		MesCP_Read					: BOOL := TRUE;	(* Read function enable *)
		MesCP_Write					: BOOL := TRUE;	(* Write function enable *)
                 
END_VAR

METHOD M_AlarmManagement
//////////////////
// Digiware measurement tool alarm and warning management
/////////////////

VAR 
	
END_VAR
END_METHOD

METHOD M_CP
//////////////////
//  Emulator
/////////////////

VAR 
	// Method local variables (reinitialized at each cycle) 
	
END_VAR
Trig_Cmd_Read(CLK:=IN_CmdToggleRead);

IF Trig_Cmd_Read.Q THEN
	IN_CmdToggleRead := FALSE;
	MesCP_Read := NOT MesCP_Read;
END_IF
END_METHOD

METHOD M_Execute
//////////////////
//  Method Calls 
/////////////////
VAR 
	// Method local variables (reinitialized at each cycle) 
	// EMULATOR

	
END_VAR
// READING AND WRITING CLOCK //
	TP1(IN:=NOT TP1.Q , PT:= ParamClockReadTime);
	ClockRead 		:= TP1.Q;

// PERMANENT CONDITIONS //
	M_CP() ; 
	
// METHODS CALLS //
	IF bInit THEN
		M_Init() ; 
		bInit					:= FALSE ; 
	ELSIF CmdInit_G OR IN_CmdReset_L THEN 
		bInit:= TRUE ;		
	END_IF

	M_Read() ; 
	M_AlarmManagement();
END_METHOD

METHOD M_Init
VAR 

END_VAR
END_METHOD

METHOD M_Read
//////////////////
//  Read Modbus Variable for PCS . 
/////////////////
VAR 
	// Method local variables (reinitialized at each cycle) 
	
END_VAR
END_METHOD

END_FUNCTION_BLOCK

// ---- 01_Equipement_Library/Operation Meter/FB_PM_A40.TcPOU
FUNCTION_BLOCK FB_PM_A40 EXTENDS FB_PM_Base
//////////////////
// Measurement Solution based on Digiware, but access through PMS Socomec
//////////////////

VAR_INPUT PERSISTENT
	// Parameters of the Object (instance specific)
	{attribute 'OPC.UA.DA' := '1'}  
	ParamUnitID					: BYTE := 22; 										// (NA) All unit ID For the Device (I35 + 1 U20)                                                                    			
	{attribute 'OPC.UA.DA' := '1'}                                                                             			
	ParamIPAddress			   	: STRING := '192.168.20.15'; 						// (NA) IP Adress of D50 .
	{attribute 'OPC.UA.DA' := '1'} 
	ParamTCPPort				: UINT := 502;										// Modbus TCP Port


END_VAR

VAR_OUTPUT
	//Child objects
	
END_VAR
VAR
	//M_ALARMMANAGEMENT VARIABLES//
		
	//M_READ VARIABLES//
		FB_ModbusRead_I1			: ARRAY[1..2] OF  FB_ModbusRead ; 				// (NA) FB for Modbus Reading
	                                                                                    	
		MesBlock1_Temp 				: ARRAY[1..2] 	OF ARRAY[0..124] OF WORD;		//(NA) Temporary Block with multiple modbus reading (U30 + I35)
		MesModbusReadAlarm 		  	: ARRAY[1..2] OF BOOL ; 						// (NA) Modbus Read Alarm for communication 
		
		
		MesModbusAlarmCode			: ARRAY[1..2] OF UDINT;							// (NA) Modbus Read Alarm Code	
		
	//M_INIT VARIABLES //
		
	// M_EXECUTE VARIABLES //
		   	MesDataExd AT %Q*			: PM_Standard ;               


 
END_VAR

METHOD M_AlarmManagement
//////////////////
// Digiware measurement tool alarm and warning management
/////////////////

VAR 
	// Method local variables (reinitialized at each cycle) 
	FB_AlarmCodeManager			: FB_AlarmCodeManager ; 
	
	KK							: BYTE ;		// For loop
	
	CMWarning					: BOOL;			// At least one Digiware device in Alarm
	CMAlarm						: BOOL;			// At least one Digiware device in Alarm
	
END_VAR
// COMMUNICATION // 

		CMWarning 		:= MesModbusReadAlarm[1] ;
		CMAlarm			:= MesModbusReadAlarm[1];
		
	// Warning
	MesWarningCom 		:= CMWarning ; 											// LOC with at least one Digiware module
	//Alarm
	TON_ComAlarm(IN:= CMAlarm, PT:= ParamTempoComAlarm, Q=>MesDataExd.MesData.MesAlarmCom) ;	 	// D50 LOC

// ALARM CODE //
	FB_AlarmCodeManager(
		bAlarm1			:=MesDataExd.MesData.MesAlarmCom , 					// Communication Alarm  #COM
		bAlarm2			:=FALSE, 									// 
		bAlarm3			:=FALSE, 									// 
		bAlarm4			:=FALSE, 									// 
		bAlarm5			:=FALSE, 									//
		bAlarm6			:=FALSE,                                    //
		bAlarm7			:=FALSE,                                    //
		bAlarm8			:=FALSE, 									//
		bAlarm9			:=FALSE,                                    //
		bAlarm10		:=FALSE,                                    //
		bAlarm11		:=FALSE, 									//
		bAlarm12		:=FALSE,                                    //
		bAlarm13		:=FALSE,                                    //
		bAlarm14		:=FALSE, 									//
		bAlarm15		:= FALSE , 									// 						 
		wAlarmCode		=>MesDataExd.MesData.MesAlarmCode);

// WARNING CODE //
	FB_AlarmCodeManager(		
		bAlarm1			:= MesWarningCom,				// Communication warning  #COM
		bAlarm2			:=FALSE, 						// 
		bAlarm3			:=FALSE, 						// 
		bAlarm4			:=FALSE, 						// 
		bAlarm5			:=FALSE, 						//
		bAlarm6			:=FALSE,                        //
		bAlarm7			:=FALSE,                        //
		bAlarm8			:=FALSE,                        //
		bAlarm9			:=FALSE,                        //
		bAlarm10		:=FALSE,                        //
		bAlarm11		:=FALSE,                        //
		bAlarm12		:=FALSE,                        //
		bAlarm13		:=FALSE,                        //
		bAlarm14		:=FALSE,                        //
		bAlarm15		:=FALSE,                        //
		wAlarmCode		=>MesDataExd.MesData.MesWarningCode);
END_METHOD

METHOD M_Read
//////////////////
//  Read Modbus Variable for PCS . 
/////////////////
VAR 
	// Method local variables (reinitialized at each cycle) 
	MW 					: FB_MergeWordsToDint; 
	KK					: BYTE;  						// FOR Loop 

	Pinterm				: REAL;
	Pinterm1			: REAL;
	Pinterm2			: REAL;
	Pinterm3			: REAL;
	Iinterm1			: REAL;
	Iinterm2			: REAL;
	Iinterm3			: REAL;
	IInterm				: REAL;
	QInterm1			: REAL;
	QInterm2			: REAL;
	QInterm3			: REAL;
	QInterm				: REAL;
	SInterm				: REAL;
END_VAR
//INITIALIZING MODBUS REQUESTS //
	FOR KK:=1 TO 2 DO
		FB_ModbusRead_I1[KK](Reset:= CmdClearFault_G ,sIPAddr:=ParamIPAddress, tTimeout:= ParamTimeout, 	nTCPport := ParamTCPPort	);
	
	END_FOR 

// CP-Read / Write 

MesDataExd.MesData.MesCP_Read := MesCP_Read ; 

IF MesCP_Read  THEN		
// MODBUS REQUEST//
	FB_ModbusRead_I1[1](
		nQuantity		:= 89, 
		nMBAddr			:= 16#4800, 
		nUnitID			:= ParamUnitID,
		cbLength		:= SIZEOF(MesBlock1_Temp[1]) , 
		pDestAddr		:= ADR(MesBlock1_Temp[1]) ,
		ClockRead		:=  MesCP_Read AND ClockRead ,
		ModbusReadAlarm	=>	MesModbusReadAlarm[1]);
		
		
		
	FB_ModbusRead_I1[2](
		nQuantity		:= 54, 
		nMBAddr			:= 16#4D80, 
		nUnitID			:= ParamUnitID,
		cbLength		:= SIZEOF(MesBlock1_Temp[2]) , 
		pDestAddr		:= ADR(MesBlock1_Temp[2]) ,
		ClockRead		:=  MesCP_Read AND ClockRead ,
		ModbusReadAlarm	=>	MesModbusReadAlarm[2]);		
		
		
// PROPERTIES UPDATE // 
	
	// Block2
	MW(WORD_STRONG:= MesBlock1_Temp[1][4], WORD_WEAK := MesBlock1_Temp[1][5],SIGNED:=FALSE, FIX:=2 , SIZE:=2, VAR_OUT := MesDataExd.MesData.MesV);	
	MW(WORD_STRONG:= MesBlock1_Temp[1][6], WORD_WEAK := MesBlock1_Temp[1][7],SIGNED:=FALSE, FIX:=2 , SIZE:=2, VAR_OUT := MesDataExd.MesData.MesU);	
	MW(WORD_STRONG:= MesBlock1_Temp[1][8], WORD_WEAK := MesBlock1_Temp[1][9],SIGNED:=FALSE, FIX:=3 , SIZE:=2, VAR_OUT := MesDataExd.MesData.MesI);	
	MW(WORD_STRONG:= MesBlock1_Temp[1][10], WORD_WEAK := MesBlock1_Temp[1][11],SIGNED:=FALSE, FIX:=3 , SIZE:=2, VAR_OUT := MesDataExd.MesData.MesFreq);	
	MW(WORD_STRONG:= MesBlock1_Temp[1][12], WORD_WEAK := MesBlock1_Temp[1][13],SIGNED:=FALSE, FIX:=2 , SIZE:=2, VAR_OUT := MesDataExd.MesData.MesV1);	
	MW(WORD_STRONG:= MesBlock1_Temp[1][14], WORD_WEAK := MesBlock1_Temp[1][15],SIGNED:=FALSE, FIX:=2 , SIZE:=2, VAR_OUT := MesDataExd.MesData.MesV2);	
	MW(WORD_STRONG:= MesBlock1_Temp[1][16], WORD_WEAK := MesBlock1_Temp[1][17],SIGNED:=FALSE, FIX:=2 , SIZE:=2, VAR_OUT := MesDataExd.MesData.MesV3);	
	MW(WORD_STRONG:= MesBlock1_Temp[1][20], WORD_WEAK := MesBlock1_Temp[1][21],SIGNED:=FALSE, FIX:=2 , SIZE:=2, VAR_OUT := MesDataExd.MesData.MesU12);	
	MW(WORD_STRONG:= MesBlock1_Temp[1][22], WORD_WEAK := MesBlock1_Temp[1][23],SIGNED:=FALSE, FIX:=2 , SIZE:=2, VAR_OUT := MesDataExd.MesData.MesU23);	
	MW(WORD_STRONG:= MesBlock1_Temp[1][24], WORD_WEAK := MesBlock1_Temp[1][25],SIGNED:=FALSE, FIX:=2 , SIZE:=2, VAR_OUT := MesDataExd.MesData.MesU31);	
	MW(WORD_STRONG:= MesBlock1_Temp[1][26], WORD_WEAK := MesBlock1_Temp[1][27],SIGNED:=FALSE, FIX:=3 , SIZE:=2, VAR_OUT := MesDataExd.MesData.MesI1);	
	MW(WORD_STRONG:= MesBlock1_Temp[1][28], WORD_WEAK := MesBlock1_Temp[1][29],SIGNED:=FALSE, FIX:=3 , SIZE:=2, VAR_OUT := MesDataExd.MesData.MesI2);	
	MW(WORD_STRONG:= MesBlock1_Temp[1][30], WORD_WEAK := MesBlock1_Temp[1][31],SIGNED:=FALSE, FIX:=3 , SIZE:=2, VAR_OUT := MesDataExd.MesData.MesI3);
	MW(WORD_STRONG:= MesBlock1_Temp[1][44], WORD_WEAK := MesBlock1_Temp[1][45],SIGNED:=TRUE, FIX:=3 , SIZE:=2, VAR_OUT := MesDataExd.MesData.MesP);	
	MW(WORD_STRONG:= MesBlock1_Temp[1][46], WORD_WEAK := MesBlock1_Temp[1][47],SIGNED:=TRUE, FIX:=3 , SIZE:=2, VAR_OUT := MesDataExd.MesData.MesQ);	
	MW(WORD_STRONG:= MesBlock1_Temp[1][52], WORD_WEAK := MesBlock1_Temp[1][53],SIGNED:=FALSE, FIX:=3 , SIZE:=2, VAR_OUT := MesDataExd.MesData.MesS);	
	MW(WORD_STRONG:= MesBlock1_Temp[1][54],SIGNED:=TRUE, FIX:=3 , SIZE:=1, VAR_OUT := MesDataExd.MesData.MesCosPhi);		
	MW(WORD_STRONG:= MesBlock1_Temp[1][56], WORD_WEAK := MesBlock1_Temp[1][57],SIGNED:=TRUE, FIX:=3 , SIZE:=2, VAR_OUT := MesDataExd.MesData.MesP1);	
	MW(WORD_STRONG:= MesBlock1_Temp[1][58], WORD_WEAK := MesBlock1_Temp[1][59],SIGNED:=TRUE, FIX:=3 , SIZE:=2, VAR_OUT := MesDataExd.MesData.MesP2);	
	MW(WORD_STRONG:= MesBlock1_Temp[1][60], WORD_WEAK := MesBlock1_Temp[1][61],SIGNED:=TRUE, FIX:=3 , SIZE:=2, VAR_OUT := MesDataExd.MesData.MesP3);	
	MW(WORD_STRONG:= MesBlock1_Temp[1][62], WORD_WEAK := MesBlock1_Temp[1][63],SIGNED:=TRUE, FIX:=3 , SIZE:=2, VAR_OUT := MesDataExd.MesData.MesQ1);	
	MW(WORD_STRONG:= MesBlock1_Temp[1][64], WORD_WEAK := MesBlock1_Temp[1][65],SIGNED:=TRUE, FIX:=3 , SIZE:=2, VAR_OUT := MesDataExd.MesData.MesQ2);	
	MW(WORD_STRONG:= MesBlock1_Temp[1][66], WORD_WEAK := MesBlock1_Temp[1][67],SIGNED:=TRUE, FIX:=3 , SIZE:=2, VAR_OUT := MesDataExd.MesData.MesQ3);		
	MW(WORD_STRONG:= MesBlock1_Temp[1][80], WORD_WEAK := MesBlock1_Temp[1][81],SIGNED:=FALSE, FIX:=3 , SIZE:=2, VAR_OUT := MesDataExd.MesData.MesS1);	
	MW(WORD_STRONG:= MesBlock1_Temp[1][82], WORD_WEAK := MesBlock1_Temp[1][83],SIGNED:=FALSE, FIX:=3 , SIZE:=2, VAR_OUT := MesDataExd.MesData.MesS2);	
	MW(WORD_STRONG:= MesBlock1_Temp[1][84], WORD_WEAK := MesBlock1_Temp[1][85],SIGNED:=FALSE, FIX:=3 , SIZE:=2, VAR_OUT := MesDataExd.MesData.MesS3);	
	MW(WORD_STRONG:= MesBlock1_Temp[1][86],SIGNED:=TRUE, FIX:=3 , SIZE:=1, VAR_OUT := MesDataExd.MesData.MesCosPhi1);	
	MW(WORD_STRONG:= MesBlock1_Temp[1][87],SIGNED:=TRUE, FIX:=3 , SIZE:=1, VAR_OUT := MesDataExd.MesData.MesCosPhi2);
	MW(WORD_STRONG:= MesBlock1_Temp[1][88],SIGNED:=TRUE, FIX:=3 , SIZE:=1, VAR_OUT := MesDataExd.MesData.MesCosPhi3);
	

	// energies 
	MW(WORD_STRONG:= MesBlock1_Temp[2][4], WORD_WEAK := MesBlock1_Temp[2][5],SIGNED:=FALSE, FIX:=4 , SIZE:=2, VAR_OUT := MesDataExd.MesData.MesEActCons);
	MW(WORD_STRONG:= MesBlock1_Temp[2][7], WORD_WEAK := MesBlock1_Temp[2][8],SIGNED:=FALSE, FIX:=4 , SIZE:=2, VAR_OUT := MesDataExd.MesData.MesEActProd);	
	MW(WORD_STRONG:= MesBlock1_Temp[2][10], WORD_WEAK := MesBlock1_Temp[2][11],SIGNED:=FALSE, FIX:=4 , SIZE:=2, VAR_OUT := MesDataExd.MesData.MesEReactCons);
	MW(WORD_STRONG:= MesBlock1_Temp[2][13], WORD_WEAK := MesBlock1_Temp[2][14],SIGNED:=FALSE, FIX:=4 , SIZE:=2, VAR_OUT := MesDataExd.MesData.MesEReactProd);
	

END_IF

// Evaluate 
	IF MesDataExd.MesData.MesP > 0.01 OR MesDataExd.MesData.MesP < -0.01 THEN
	MesDataExd.MesData.MesTanPhi := MesDataExd.MesData.MesQ /MesDataExd.MesData.MesP;
	ELSE
	MesDataExd.MesData.MesTanPhi := 0;
	END_IF
END_METHOD

END_FUNCTION_BLOCK

// ---- 01_Equipement_Library/Operation Meter/FB_PM_Digiware.TcPOU
FUNCTION_BLOCK FB_PM_Digiware EXTENDS FB_PM_Base
//////////////////
// Measurement Solution based on Digiware, but access through PMS Socomec
//////////////////

VAR_INPUT PERSISTENT
	// Parameters of the Object (instance specific) 
	ParamUnitID					: BYTE	 	;						// (NA) U30 unit ID
	ParamIPAddress			   	: STRING 	;							// (NA) IP Adress of D50 .
	ParamTCPPort				: UINT 		;
	ParamInvertPower			: BOOL		;
END_VAR

VAR_OUTPUT
	//Child objects
	
END_VAR
VAR
	//M_ALARMMANAGEMENT VARIABLES//
		
	//M_READ VARIABLES//
		MesDataExd					: PM_DirisA40;
		
		ModbusRead					: ARRAY[1..5] OF FB_ModbusRead ; 			// (NA) FB for Modbus Reading
		MesBlock1_Temp 				: ARRAY[1..5] OF ARRAY[1..120] OF WORD;		//(NA) Temporary Block with multiple modbus reading (U30 + I35)
		
		
	//M_CP VARIABLES //
		CmdWrite						: BOOL;
		Trig_Read						: R_TRIG;
		Trig_Write						: R_TRIG;

	// M_EXECUTE VARIABLES //

 
END_VAR

METHOD M_AlarmManagement
//////////////////
// Digiware measurement tool alarm and warning management
/////////////////

VAR 
	// Method local variables (reinitialized at each cycle) 
	FB_AlarmCodeManager			: FB_AlarmCodeManager ; 
	
	KK							: BYTE ;		// For loop
	
	
END_VAR
IF MesDataExd.MesData.MesCP_Read THEN
// COMMUNICATION // 
	TON_ComWarning(PT := ParamTempoComAlarm, IN := ModbusRead[1].ModbusReadAlarm OR ModbusRead[2].ModbusReadAlarm OR ModbusRead[3].ModbusReadAlarm) ; 											// LOC with at least one Digiware module
	TON_ComAlarm(PT := ParamTempoComAlarm, IN := ModbusRead[1].ModbusReadAlarm AND ModbusRead[2].ModbusReadAlarm AND ModbusRead[3].ModbusReadAlarm)	 ; 											// LOC with at least one Digiware module
ELSE
	TON_ComWarning(IN := FALSE);
	TON_ComAlarm(IN := FALSE);
END_IF

MesDataExd.MesComAlarm 	:= TON_ComAlarm.Q;
MesDataExd.MesComWarning 	:= TON_ComWarning.Q;

// ALARM CODE //
	FB_AlarmCodeManager(
		bAlarm1			:= MesDataExd.MesComAlarm, 			// Communication Error : All Modbus TCP Frame failed
		bAlarm2			:=FALSE, 							// 
		bAlarm3			:=FALSE, 							// 
		bAlarm4			:=FALSE, 							// 
		bAlarm5			:=FALSE, 							//  			
		bAlarm6			:=FALSE,  							// 
		bAlarm7			:=FALSE,  							// 
		bAlarm8			:=FALSE,  							// 
		bAlarm9			:=FALSE,  							// 
		bAlarm10		:=FALSE,  							// 
		bAlarm11		:=FALSE,  							// 
		bAlarm12		:=FALSE,  							// 
		bAlarm13		:=FALSE,  							// 
		bAlarm14		:=FALSE,  							// 
		bAlarm15		:=False , 							// 					 
		wAlarmCode		=> MesDataExd.MesData.MesAlarmCode);

// WARNING CODE //
	FB_AlarmCodeManager(		
		bAlarm1			:= MesDataExd.MesComWarning,				 	// Communication Warning : At least one Modbus TCP Frame failed
		bAlarm2			:=FALSE, 							// 
		bAlarm3			:=FALSE, 							// 
		bAlarm4			:=FALSE, 							// 
		bAlarm5			:=FALSE,  							// 
		bAlarm6			:=FALSE,  							// 
		bAlarm7			:=FALSE,  							// 
		bAlarm8			:=FALSE,  							// 
		bAlarm9			:=FALSE,  							// 
		bAlarm10		:=FALSE,  							// 
		bAlarm11		:=FALSE,  							// 
		bAlarm12		:=FALSE,  							// 
		bAlarm13		:=FALSE,  							// 
		bAlarm14		:=FALSE,  							// 
		bAlarm15		:=FALSE,  							// 
		wAlarmCode		=> MesDataExd.MesData.MesWarningCode);
END_METHOD

METHOD M_CP 
VAR_INPUT
END_VAR

IF IN_CmdToggleRead THEN
	IN_CmdToggleRead := FALSE;
	MesDataExd.MesData.MesCP_Read := NOT MesDataExd.MesData.MesCP_Read;
END_IF
END_METHOD

METHOD M_Init
VAR 

	KK: BYTE;
END_VAR
ParamTCPPort			:= 502;

MesDataExd.MesData.MesCP_Read := TRUE;
END_METHOD

METHOD M_Read
//////////////////
//  Read Modbus Variable for PCS . 
/////////////////
VAR 
	// Method local variables (reinitialized at each cycle) 
	MW 					: FB_MergeWordsToDint; 
	KK					: BYTE;  						// FOR Loop 

	AX_ADDR				: ARRAY[1.. 5] OF UINT := [50514, 	50780, 	51536];
	AX_QTY				: ARRAY[1.. 5] OF BYTE := [78,		46,		10];
	AX_UnitId			: ARRAY[1.. 5] OF BYTE := [1,		1,		1];
	
END_VAR
FOR KK := 1 TO 3 DO
	ModbusRead[KK]
	(
		sIPAddr := ParamIPAddress,
		pDestAddr := ADR(MesBlock1_Temp[KK]),
		tTimeout := ParamTimeout,
		nTcpPort := ParamTCPPort,
		nQuantity := AX_QTY[KK],
		cbLength := SIZEOF(MesBlock1_Temp[KK]),
		nUnitID := ParamUnitID,
		nMBAddr := AX_ADDR[KK],
		ClockRead := ClockRead AND MesDataExd.MesData.MesCP_Read
	);
END_FOR

	IF MesDataExd.MesData.MesCP_Read THEN
	// PROPERTIES UPDATE // 
		// Block 1
		 	MW(WORD_STRONG:= MesBlock1_Temp[1][ 1], WORD_WEAK := MesBlock1_Temp[1][ 2],	SIGNED:=FALSE, 	FIX:=2 , SIZE:=2, VAR_OUT:=MesDataExd.MesData.MesU12);
			MW(WORD_STRONG:= MesBlock1_Temp[1][ 3], WORD_WEAK := MesBlock1_Temp[1][ 4],	SIGNED:=FALSE, 	FIX:=2 , SIZE:=2, VAR_OUT:=MesDataExd.MesData.MesU23);
			MW(WORD_STRONG:= MesBlock1_Temp[1][ 5], WORD_WEAK := MesBlock1_Temp[1][ 6],	SIGNED:=FALSE, 	FIX:=2 , SIZE:=2, VAR_OUT:=MesDataExd.MesData.MesU31);
			MW(WORD_STRONG:= MesBlock1_Temp[1][ 7], WORD_WEAK := MesBlock1_Temp[1][ 8],	SIGNED:=FALSE, 	FIX:=2 , SIZE:=2, VAR_OUT:=MesDataExd.MesData.MesV1);
			MW(WORD_STRONG:= MesBlock1_Temp[1][ 9], WORD_WEAK := MesBlock1_Temp[1][10],	SIGNED:=FALSE, 	FIX:=2 , SIZE:=2, VAR_OUT:=MesDataExd.MesData.MesV2);
			MW(WORD_STRONG:= MesBlock1_Temp[1][11], WORD_WEAK := MesBlock1_Temp[1][12],	SIGNED:=FALSE, 	FIX:=2 , SIZE:=2, VAR_OUT:=MesDataExd.MesData.MesV3);
			MW(WORD_STRONG:= MesBlock1_Temp[1][13], WORD_WEAK := MesBlock1_Temp[1][14],	SIGNED:=FALSE, 	FIX:=2 , SIZE:=2, VAR_OUT:=MesDataExd.MesData.MesFreq);
			MW(WORD_STRONG:= MesBlock1_Temp[1][15], WORD_WEAK := MesBlock1_Temp[1][16],	SIGNED:=FALSE, 	FIX:=3 , SIZE:=2, VAR_OUT:=MesDataExd.Mesdata.MesI1);
			MW(WORD_STRONG:= MesBlock1_Temp[1][17], WORD_WEAK := MesBlock1_Temp[1][18],	SIGNED:=FALSE, 	FIX:=3 , SIZE:=2, VAR_OUT:=MesDataExd.Mesdata.MesI2);
			MW(WORD_STRONG:= MesBlock1_Temp[1][19], WORD_WEAK := MesBlock1_Temp[1][20],	SIGNED:=FALSE, 	FIX:=3 , SIZE:=2, VAR_OUT:=MesDataExd.Mesdata.MesI3);
			MW(WORD_STRONG:= MesBlock1_Temp[1][21], WORD_WEAK := MesBlock1_Temp[1][22],	SIGNED:=FALSE, 	FIX:=3 , SIZE:=2, VAR_OUT:=MesDataExd.Mesdata.mesIn);
			MW(WORD_STRONG:= MesBlock1_Temp[1][23], WORD_WEAK := MesBlock1_Temp[1][24],	SIGNED:=TRUE, 	FIX:=2 , SIZE:=2, VAR_OUT:=MesDataExd.Mesdata.mesP);
			MW(WORD_STRONG:= MesBlock1_Temp[1][25], WORD_WEAK := MesBlock1_Temp[1][26],	SIGNED:=TRUE, 	FIX:=2 , SIZE:=2, VAR_OUT:=MesDataExd.Mesdata.mesQ);
			MW(WORD_STRONG:= MesBlock1_Temp[1][27], WORD_WEAK := MesBlock1_Temp[1][28],	SIGNED:=FALSE, 	FIX:=2 , SIZE:=2, VAR_OUT:=MesDataExd.Mesdata.mesS);
			MW(WORD_STRONG:= MesBlock1_Temp[1][29], WORD_WEAK := MesBlock1_Temp[1][30],	SIGNED:=TRUE, 	FIX:=3 , SIZE:=2, VAR_OUT:=MesDataExd.Mesdata.MesCosPhi);
			MW(WORD_STRONG:= MesBlock1_Temp[1][31], WORD_WEAK := MesBlock1_Temp[1][32],	SIGNED:=TRUE, 	FIX:=2 , SIZE:=2, VAR_OUT:=MesDataExd.Mesdata.MesP1);
			MW(WORD_STRONG:= MesBlock1_Temp[1][33], WORD_WEAK := MesBlock1_Temp[1][34],	SIGNED:=TRUE, 	FIX:=2 , SIZE:=2, VAR_OUT:=MesDataExd.Mesdata.MesP2);
			MW(WORD_STRONG:= MesBlock1_Temp[1][35], WORD_WEAK := MesBlock1_Temp[1][36],	SIGNED:=TRUE, 	FIX:=2 , SIZE:=2, VAR_OUT:=MesDataExd.Mesdata.MesP3);
			MW(WORD_STRONG:= MesBlock1_Temp[1][37], WORD_WEAK := MesBlock1_Temp[1][38],	SIGNED:=TRUE, 	FIX:=2 , SIZE:=2, VAR_OUT:=MesDataExd.Mesdata.MesQ1);
			MW(WORD_STRONG:= MesBlock1_Temp[1][39], WORD_WEAK := MesBlock1_Temp[1][40],	SIGNED:=TRUE, 	FIX:=2 , SIZE:=2, VAR_OUT:=MesDataExd.Mesdata.MesQ2);
			MW(WORD_STRONG:= MesBlock1_Temp[1][41], WORD_WEAK := MesBlock1_Temp[1][42],	SIGNED:=TRUE, 	FIX:=2 , SIZE:=2, VAR_OUT:=MesDataExd.Mesdata.MesQ3);
			
		
		
		// Block2
			MW(WORD_STRONG:= MesBlock1_Temp[2][ 1], WORD_WEAK := MesBlock1_Temp[2][ 2], SIGNED:=FALSE, FIX:=0 , SIZE:=1, VAR_OUT:=MesDataExd.MesData.MesEActProd);
			MW(WORD_STRONG:= MesBlock1_Temp[2][ 3], WORD_WEAK := MesBlock1_Temp[2][ 4], SIGNED:=FALSE, FIX:=0 , SIZE:=1, VAR_OUT:=MesDataExd.MesData.MesEReactProd);
			MW(WORD_STRONG:= MesBlock1_Temp[2][ 7], WORD_WEAK := MesBlock1_Temp[2][ 8], SIGNED:=FALSE, FIX:=0 , SIZE:=1, VAR_OUT:=MesDataExd.MesData.MesEActCons);
			MW(WORD_STRONG:= MesBlock1_Temp[2][ 9], WORD_WEAK := MesBlock1_Temp[2][10], SIGNED:=FALSE, FIX:=0 , SIZE:=1, VAR_OUT:=MesDataExd.MesData.MesEReactCons);
		
		// Block3
			MW(WORD_STRONG:= MesBlock1_Temp[3][ 1], SIGNED:=FALSE, FIX:=2 , SIZE:=1, VAR_OUT:=MesDataExd.MesTHDU12);
			MW(WORD_STRONG:= MesBlock1_Temp[3][ 2], SIGNED:=FALSE, FIX:=2 , SIZE:=1, VAR_OUT:=MesDataExd.MesTHDU23);
			MW(WORD_STRONG:= MesBlock1_Temp[3][ 3], SIGNED:=FALSE, FIX:=2 , SIZE:=1, VAR_OUT:=MesDataExd.MesTHDU31);
			MW(WORD_STRONG:= MesBlock1_Temp[3][ 4], SIGNED:=FALSE, FIX:=2 , SIZE:=1, VAR_OUT:=MesDataExd.MesTHDV1);
			MW(WORD_STRONG:= MesBlock1_Temp[3][ 5], SIGNED:=FALSE, FIX:=2 , SIZE:=1, VAR_OUT:=MesDataExd.MesTHDV2);
			MW(WORD_STRONG:= MesBlock1_Temp[3][ 6], SIGNED:=FALSE, FIX:=2 , SIZE:=1, VAR_OUT:=MesDataExd.MesTHDV3);
			MW(WORD_STRONG:= MesBlock1_Temp[3][ 7], SIGNED:=FALSE, FIX:=2 , SIZE:=1, VAR_OUT:=MesDataExd.MesTHDI1);
			MW(WORD_STRONG:= MesBlock1_Temp[3][ 8], SIGNED:=FALSE, FIX:=2 , SIZE:=1, VAR_OUT:=MesDataExd.MesTHDI2);
			MW(WORD_STRONG:= MesBlock1_Temp[3][ 9], SIGNED:=FALSE, FIX:=2 , SIZE:=1, VAR_OUT:=MesDataExd.MesTHDI3);
			MW(WORD_STRONG:= MesBlock1_Temp[3][10], SIGNED:=FALSE, FIX:=2 , SIZE:=1, VAR_OUT:=MesDataExd.MesTHDIN);
			
		MesDataExd.MesData.MesI := (MesDataExd.Mesdata.MesI1 + MesDataExd.MesData.MesI2 + MesDataExd.MesData.mesI3)/3;
		MesDataExd.MesData.MesU := (MesDataExd.Mesdata.MesU12 + MesDataExd.MesData.MesU23 + MesDataExd.MesData.mesU31)/3;
		MesDataExd.MesData.MesV := (MesDataExd.MesData.MesV1 + MesDataExd.MesData.MesV2 + MesDataExd.mesdata.MesV3)/3;
		IF ParamInvertPower THEN
			MesDataExd.MesData.MesP 	:= - MesDataExd.MesData.MesP;
			MesDataExd.MesData.MesP1 	:= - MesDataExd.MesData.MesP1;
			MesDataExd.MesData.MesP2 	:= - MesDataExd.MesData.MesP2;
			MesDataExd.MesData.MesP3 	:= - MesDataExd.MesData.MesP3;
			MesDataExd.MesData.MesQ 	:= - MesDataExd.MesData.MesQ;
			MesDataExd.MesData.MesQ1 	:= - MesDataExd.MesData.MesQ1;
			MesDataExd.MesData.MesQ2 	:= - MesDataExd.MesData.MesQ2;
			MesDataExd.MesData.MesQ3 	:= - MesDataExd.MesData.MesQ3;
		END_IF
	END_IF
END_METHOD

END_FUNCTION_BLOCK

// ---- 01_Equipement_Library/Operation Meter/FB_PM_ION7650.TcPOU
FUNCTION_BLOCK FB_PM_ION7650 EXTENDS FB_PM_Base
//////////////////
// Measurement Solution based on Digiware, but access through PMS Socomec
//////////////////
VAR CONSTANT
	// Characteristics of the object (Same for all instances)
			
END_VAR

VAR_INPUT PERSISTENT
	// Parameters of the Object (instance specific) 
	{attribute 'OPC.UA.DA' := '1'} 
	ParamUnitID					: BYTE 		:= 1 ;								(* (NA) Unit ID*)
//	ParamInInterfaceSub			: BOOL 		:= TRUE; 							// (NA) Serial interface RS422/RS485 TYPE (0:EL6021,1:SUB9)
	{attribute 'OPC.UA.DA' := '1'} 
	ParamIPAdress		   		: STRING 	:= '192.168.20.15'; 				(* (NA) IP Adress of ION7650 *)
	{attribute 'OPC.UA.DA' := '1'} 
	ParamTcpPort				: UINT 		:= 502;								(* (NA) TCP port			*)
	ParamPCountZero				: INT		:= 1;								(* (NA) Number of time the PM P measurement was reinitialized to zero *)

END_VAR

VAR_OUTPUT
	//Child objects
	
END_VAR
VAR                                                  								                                          								
	//M_READ VARIABLES//
		FB_ModbusRead				: FB_ModbusRTU ;						// (NA) FB for Modbus Reading
		InputStructRead 			: ARRAY[1..1] OF  Struct_InputRTU;
		
		AX_Quantity					: ARRAY[1..1] OF WORD;					// (NA) Quantity of blocks to read
		AX_Address					: ARRAY[1..1] OF WORD;					// (NA) Start address of the read
		MesBlock_Temp 				: ARRAY[1..1] OF ARRAY[1..125] OF WORD;	// (NA) Temporary Block with multiple modbus reading (U30 + I35)
		Busy						: BOOL;
		OutErrorMbRead				: ARRAY[1..1] OF BOOL;
		
		RTrigI						: R_TRIG;
	//M_INIT VARIABLES //
		OutFBCompleteted			: BOOL;
	// ION was reset to 0 
		IONCount_PossibleReset		: BOOL := TRUE; 						// (NA) The active power of the PM ION7650 is between 1000 and  10m 
		
		
	MesDataExd AT %Q*				: PM_Standard ;
		
END_VAR

METHOD M_AlarmManagement
//////////////////
// Digiware measurement tool alarm and warning management
/////////////////

VAR 
	// Method local variables (reinitialized at each cycle) 
	FB_AlarmCodeManager			: FB_AlarmCodeManager ; 
	
	KK							: BYTE ;		// For loop
	
	CMWarning					: BOOL;			// At least one Digiware device in Alarm
	CMAlarm						: BOOL;			// At least one Digiware device in Alarm
	
END_VAR
TON_ComAlarm(IN:= OutErrorMbRead[1], PT:= ParamTempoComAlarm, Q=>MesDataExd.MesData.MesAlarmCom) ;	
//					General com alarm : All the read FB fucked up

// ALARM CODE //
	FB_AlarmCodeManager( 
		bAlarm1			:=MesDataExd.MesData.MesAlarmCom, 					// Communication Error  #COM
		bAlarm2			:=FALSE, 									// 
		bAlarm3			:=FALSE, 									// 
		bAlarm4			:=FALSE, 									// 
		bAlarm5			:=FALSE, 									//
		bAlarm6			:=FALSE, 									//
		bAlarm7			:=FALSE, 									//
		bAlarm8			:=FALSE, 									//
		bAlarm9			:=FALSE, 									//
		bAlarm10		:=FALSE, 									//
		bAlarm11		:=FALSE, 									//
		bAlarm12		:=FALSE, 									//
		bAlarm13		:=FALSE, 									//
		bAlarm14		:=FALSE, 									//
		bAlarm15		:= FALSE , 									//						 
		wAlarmCode		=>MesDataExd.MesData.MesAlarmCode);

// WARNING CODE //
	FB_AlarmCodeManager(		
		bAlarm1			:=	MesWarningCom,				 			// Communication Warning #COM	
		bAlarm2			:=FALSE, 									// 
		bAlarm3			:=FALSE, 									// 
		bAlarm4			:=FALSE, 									// 
		bAlarm5			:=FALSE, 									//
		bAlarm6			:=FALSE, 									//
		bAlarm7			:=FALSE, 									//
		bAlarm8			:=FALSE, 									//
		bAlarm9			:=FALSE, 									//
		bAlarm10		:=FALSE, 									//
		bAlarm11		:=FALSE, 									//
		bAlarm12		:=FALSE, 									//
		bAlarm13		:=FALSE, 									//
		bAlarm14		:=FALSE, 									//
		bAlarm15		:=FALSE, 									//
		wAlarmCode		=>MesDataExd.MesData.MesWarningCode);
END_METHOD

METHOD M_Evaluate : BOOL
VAR_INPUT
END_VAR
END_METHOD

METHOD M_Init
VAR 

END_VAR
(*FB_ModbusRead(InTimeout:= ParamTimeout,
				 InUnitID:= DINT_TO_BYTE(ParamUnitID),
				 InQuantity:= 125,	
				 InInterfaceSub:= ParamInInterfaceSub,
				 InFunctionRead := FALSE);
*)
	
AX_Quantity[1] := 125;
AX_Address[1]  := 149;
END_METHOD

METHOD M_Read
//////////////////
//  Read Modbus Variable for ION7650. 
/////////////////
VAR 
	// Method local variables (reinitialized at each cycle) 
	MW 					: FB_MergeWordsToDint; 
	KK					: BYTE;  						// FOR Loop 

END_VAR
// CP-Read / Write 

MesDataExd.MesData.MesCP_Read := MesCP_Read ; 
 

IF MesCP_Read  THEN	
// MODBUS REQUEST TCP-IP //
(*	 
	ModbusRead
	(
		pDestAddr := ADR(MesBlock1_Temp),
		sIPAddr := ParamIPAdress,
		tTimeout := ParamTimeout,
		nQuantity := 122,
		nMBAddr := 150,
		cbLength := SIZEOF(MesBlock1_Temp),
		nUnitID := ParamUnitID,
		ClockRead := ClockRead,
		ErrorId => ModbusAlarmsID,
		ModbusReadAlarm => ModbusAlarm
	);
	*)
// MODBUS REQUEST RTU //	
	FB_ModbusRead();

	RTrigI(CLK:= ClockRead );
//Metrology
	FOR KK:=1 TO 1 DO
		InputStructRead[KK].InBuffer := ADR(MesBlock_Temp[KK]);
		InputStructRead[KK].InFunction := 3;
		InputStructRead[KK].InQuantity := AX_Quantity[KK];
		InputStructRead[KK].InStartAddr := AX_Address[KK];
		InputStructRead[KK].InUnitID := ParamUnitID;
		
		InputStructRead[KK].OutBusy := ADR(Busy);
		InputStructRead[KK].OutError := ADR(OutErrorMbRead[KK]);
		//InputStructRead[KK].OutCompleted := ADR(bReadCompleted);
		
		IF RTrigI.Q THEN 
			FB_ModbusRead.M_AddAction_FIFO(InStruct:= InputStructRead[KK] , InPriority:=1 ) ; 
		END_IF
		
	END_FOR 
				
// PROPERTIES UPDATE // 
	// Block 1
	MW(WORD_STRONG:= MesBlock_Temp[1][  1], SIGNED:=FALSE, FIX:=1 , SIZE:=1, 	VAR_OUT	:= MesDataExd.MesData.MesI1);
	MW(WORD_STRONG:= MesBlock_Temp[1][  2], SIGNED:=FALSE, FIX:=1 , SIZE:=1, 	VAR_OUT	:= MesDataExd.MesData.MesI2);
	MW(WORD_STRONG:= MesBlock_Temp[1][  3], SIGNED:=FALSE, FIX:=1 , SIZE:=1, 	VAR_OUT	:= MesDataExd.MesData.MesI3);
	MW(WORD_STRONG:= MesBlock_Temp[1][  6], SIGNED:=FALSE, FIX:=1 , SIZE:=1, 	VAR_OUT	:= MesDataExd.MesData.MesI);
	MW(WORD_STRONG:= MesBlock_Temp[1][ 10], SIGNED:=FALSE, FIX:=1 , SIZE:=1, 	VAR_OUT	:= MesDataExd.MesData.MesFreq);
	MW(WORD_STRONG:= MesBlock_Temp[1][ 17], Word_WEAK:= MesBlock_Temp[1][ 18], 	SIGNED:=FALSE, FIX:=0 , SIZE:=2, VAR_OUT:= MesDataExd.MesData.MesV1);
	MW(WORD_STRONG:= MesBlock_Temp[1][ 19], Word_WEAK:= MesBlock_Temp[1][ 20], 	SIGNED:=FALSE, FIX:=0 , SIZE:=2, VAR_OUT:= MesDataExd.MesData.MesV2);
	MW(WORD_STRONG:= MesBlock_Temp[1][ 21], Word_WEAK:= MesBlock_Temp[1][ 22], 	SIGNED:=FALSE, FIX:=0 , SIZE:=2, VAR_OUT:= MesDataExd.MesData.MesV3);
	MW(WORD_STRONG:= MesBlock_Temp[1][ 23], Word_WEAK:= MesBlock_Temp[1][ 24], 	SIGNED:=FALSE, FIX:=0 , SIZE:=2, VAR_OUT:= MesDataExd.MesData.MesV);
	MW(WORD_STRONG:= MesBlock_Temp[1][ 29], Word_WEAK:= MesBlock_Temp[1][ 30], 	SIGNED:=FALSE, FIX:=0 , SIZE:=2, VAR_OUT:= MesDataExd.MesData.MesU12);
	MW(WORD_STRONG:= MesBlock_Temp[1][ 31], Word_WEAK:= MesBlock_Temp[1][ 32], 	SIGNED:=FALSE, FIX:=0 , SIZE:=2, VAR_OUT:= MesDataExd.MesData.MesU23);
	MW(WORD_STRONG:= MesBlock_Temp[1][ 33], Word_WEAK:= MesBlock_Temp[1][ 34], 	SIGNED:=FALSE, FIX:=0 , SIZE:=2, VAR_OUT:= MesDataExd.MesData.MesU31);
	MW(WORD_STRONG:= MesBlock_Temp[1][ 35], Word_WEAK:= MesBlock_Temp[1][ 36], 	SIGNED:=FALSE, FIX:=0 , SIZE:=2, VAR_OUT:= MesDataExd.MesData.MesU);	
	MW(WORD_STRONG:= MesBlock_Temp[1][ 49], Word_WEAK:= MesBlock_Temp[1][ 50], 	SIGNED:=TRUE , FIX:=0 , SIZE:=2, VAR_OUT:= MesDataExd.MesData.MesP1);
	MW(WORD_STRONG:= MesBlock_Temp[1][ 51], Word_WEAK:= MesBlock_Temp[1][ 52], 	SIGNED:=TRUE , FIX:=0 , SIZE:=2, VAR_OUT:= MesDataExd.MesData.MesP2);
	MW(WORD_STRONG:= MesBlock_Temp[1][ 53], Word_WEAK:= MesBlock_Temp[1][ 54], 	SIGNED:=TRUE , FIX:=0 , SIZE:=2, VAR_OUT:= MesDataExd.MesData.MesP3);
	MW(WORD_STRONG:= MesBlock_Temp[1][ 55], Word_WEAK:= MesBlock_Temp[1][ 56], 	SIGNED:=TRUE , FIX:=0 , SIZE:=2, VAR_OUT:= MesDataExd.MesData.MesP);	
	MW(WORD_STRONG:= MesBlock_Temp[1][ 59], Word_WEAK:= MesBlock_Temp[1][ 60], 	SIGNED:=TRUE , FIX:=0 , SIZE:=2, VAR_OUT:= MesDataExd.MesData.MesQ1);	
	MW(WORD_STRONG:= MesBlock_Temp[1][ 61], Word_WEAK:= MesBlock_Temp[1][ 62], 	SIGNED:=TRUE , FIX:=0 , SIZE:=2, VAR_OUT:= MesDataExd.MesData.MesQ2);	
	MW(WORD_STRONG:= MesBlock_Temp[1][ 63], Word_WEAK:= MesBlock_Temp[1][ 64], 	SIGNED:=TRUE , FIX:=0 , SIZE:=2, VAR_OUT:= MesDataExd.MesData.MesQ3);	
	MW(WORD_STRONG:= MesBlock_Temp[1][ 65], Word_WEAK:= MesBlock_Temp[1][ 66], 	SIGNED:=TRUE , FIX:=0 , SIZE:=2, VAR_OUT:= MesDataExd.MesData.MesQ);	
	MW(WORD_STRONG:= MesBlock_Temp[1][ 75], Word_WEAK:= MesBlock_Temp[1][ 76], 	SIGNED:=TRUE , FIX:=0 , SIZE:=2, VAR_OUT:= MesDataExd.MesData.MesS);	
	                                                                                                                       
	MW(WORD_STRONG:= MesBlock_Temp[1][ 81], Word_weak:= MesBlock_Temp[1][ 82], 	SIGNED:=TRUE , FIX:=0 , SIZE:=2, VAR_OUT:= MesDataExd.MesData.MesEActProd);
	MW(WORD_STRONG:= MesBlock_Temp[1][ 83], Word_weak:= MesBlock_Temp[1][ 84], 	SIGNED:=TRUE , FIX:=0 , SIZE:=2, VAR_OUT:= MesDataExd.MesData.MesEActCons);
	MW(WORD_STRONG:= MesBlock_Temp[1][ 85], Word_weak:= MesBlock_Temp[1][ 86], 	SIGNED:=TRUE , FIX:=0 , SIZE:=2, VAR_OUT:= MesDataExd.MesData.MesEReactProd);
	MW(WORD_STRONG:= MesBlock_Temp[1][ 87], Word_weak:= MesBlock_Temp[1][ 88], 	SIGNED:=TRUE , FIX:=0 , SIZE:=2, VAR_OUT:= MesDataExd.MesData.MesEReactCons);
	                                                                 
	MW(WORD_STRONG:= MesBlock_Temp[1][113], SIGNED:=FALSE , FIX:=4 , SIZE:=1,	VAR_OUT:= MesDataExd.MesData.MesCosPhi1);
	MW(WORD_STRONG:= MesBlock_Temp[1][114], SIGNED:=FALSE , FIX:=4 , SIZE:=1,	VAR_OUT:= MesDataExd.MesData.MesCosPhi2);
	MW(WORD_STRONG:= MesBlock_Temp[1][115], SIGNED:=FALSE , FIX:=4 , SIZE:=1,	VAR_OUT:= MesDataExd.MesData.MesCosPhi3);
	MW(WORD_STRONG:= MesBlock_Temp[1][116], SIGNED:=FALSE , FIX:=4 , SIZE:=1,	VAR_OUT:= MesDataExd.MesData.MesCosPhi);
	
	
// Add the previous produced energy before counter reset
	IF MesDataExd.MesData.MesEActProd > 0 AND MesDataExd.MesData.MesEActProd < 1000  AND IONCount_PossibleReset THEN  
		IONCount_PossibleReset := FALSE;
		ParamPCountZero := ParamPCountZero + 1;	
	ELSIF MesDataExd.MesData.MesEActProd > 1000 THEN
		IONCount_PossibleReset := TRUE;
	END_IF

MesDataExd.MesData.MesEActProd := MesDataExd.MesData.MesEActProd + 10000000*ParamPCountZero;	
		
	IF MesDataExd.MesData.MesP<0.01 AND MesDataExd.MesData.MesP>-0.01  THEN 
		MesDataExd.MesData.MesTanPhi := 0 ;  
	ELSE
		MesDataExd.MesData.MesTanPhi := MesDataExd.MesData.MesQ /MesDataExd.MesData.MesP ; 
	END_IF
	
END_IF
END_METHOD

END_FUNCTION_BLOCK

// ---- 01_Equipement_Library/Operation Meter/FB_PM_Janitza.TcPOU
FUNCTION_BLOCK FB_PM_Janitza EXTENDS FB_PM_Base
//////////////////
// Measurement Solution based on Janitza, but access through JemaPLC
//////////////////

VAR_INPUT PERSISTENT
	// Parameters of the Object (instance specific) 
	{attribute 'OPC.UA.DA' := '1'} 
	ParamIpAddress			   	: STRING 		:= '192.168.1.30'; 			(* (NA) IP Adress of D50 .*)
	{attribute 'OPC.UA.DA' := '1'} 
	ParamUnitID 				: BYTE  := 1; 			  					(* (NA)   Modbus Unit ID.	*)


END_VAR

VAR_OUTPUT
	//Child objects
	
END_VAR
VAR
	//M_ALARMMANAGEMENT VARIABLES//
	
	//M_READ VARIABLES//
		FB_ModbusRead_I1			: ARRAY[1..1] OF  FB_ModbusRead ; 		// (NA) FB for Modbus Reading
	
		MesBlock1_Temp 				: ARRAY[0..125] OF WORD;				//(NA) Temporary Block with multiple modbus reading (U30 + I35)
		
		MesModbusReadAlarm 		  	: ARRAY[1..1] OF BOOL ; 				// (NA) Modbus Read Alarm for communication 
		
		MesModbusAlarmCode			: UDINT;								// (NA) Modbus Read Alarm Code	
		
	//M_INIT VARIABLES //

	// M_EXECUTE VARIABLES //
			MesDataExd AT %Q*				: PM_Standard ;
	
END_VAR

METHOD M_AlarmManagement
//////////////////
// Digiware measurement tool alarm and warning management
/////////////////

VAR 
	// Method local variables (reinitialized at each cycle) 
	FB_AlarmCodeManager			: FB_AlarmCodeManager ; 
	
	KK							: BYTE ;		// For loop
	
	CMWarning					: BOOL;			// At least one Digiware device in Alarm
	CMAlarm						: BOOL;			// At least one Digiware device in Alarm
	
END_VAR
// COMMUNICATION // 
IF MesDataExd.MesData.MesCP_Read then
	CMWarning 			:= FALSE ;
	CMAlarm	 			:= TRUE ;
	
	FOR KK:=1 TO 1 DO
		CMWarning 		:= CMWarning OR MesModbusReadAlarm[KK] ;
		CMAlarm			:= CMAlarm AND MesModbusReadAlarm[KK] ; 
	END_FOR
END_IF
	
	// Warning
	MesWarningCom 		:= CMWarning ; 											// LOC with at least one Digiware module
	//Alarm
	TON_ComAlarm(IN:= CMAlarm , PT:= ParamTempoComAlarm, Q=>MesDataExd.MesData.MesAlarmCom) ;	 	// D50 LOC

// ALARM CODE //
	FB_AlarmCodeManager(
		bAlarm1			:= MesDataExd.MesData.MesAlarmCom  , 					// Communication Alarm  #COM
		bAlarm2			:=FALSE, 		                            // 
		bAlarm3			:=FALSE, 		                            // 
		bAlarm4			:=FALSE, 		                            // 
		bAlarm5			:=FALSE,                                    //
		bAlarm6			:=FALSE,                                    //
		bAlarm7			:=FALSE,                                    //
		bAlarm8			:=FALSE,                                    //
		bAlarm9			:=FALSE,                                    //
		bAlarm10		:=FALSE,                                    //
		bAlarm11		:=FALSE,                                    //
		bAlarm12		:=FALSE,                                    //
		bAlarm13		:=FALSE,                                    //
		bAlarm14		:=FALSE,                                    //
		bAlarm15		:= FALSE , 			 						// 						 	 
		wAlarmCode		=>MesDataExd.MesData.MesAlarmCode);

// WARNING CODE //
	FB_AlarmCodeManager(		
		bAlarm1			:= MesWarningCom	,				// Communication warning  #COM
		bAlarm2			:=FALSE, 		                 	// 
		bAlarm3			:=FALSE, 		                  	// 
		bAlarm4			:=FALSE, 		                 	// 
		bAlarm5			:=FALSE,                            //
		bAlarm6			:=FALSE,                            //
		bAlarm7			:=FALSE,                            //
		bAlarm8			:=FALSE,                            //
		bAlarm9			:=FALSE,                            //
		bAlarm10		:=FALSE,                            //
		bAlarm11		:=FALSE,                            //
		bAlarm12		:=FALSE,                            //
		bAlarm13		:=FALSE,                            //
		bAlarm14		:=FALSE,                            //
		bAlarm15		:=FALSE,                            //
		wAlarmCode		=>MesDataExd.MesData.MesWarningCode);
END_METHOD

METHOD M_Read
//////////////////
//  Read Modbus Variable for PCS . 
/////////////////
VAR 
	// Method local variables (reinitialized at each cycle) 
	MW 			: FB_MergeWordsToFloat ;
	
	MesPW	 : REAL ; 
	MesP1W   : REAL ; 
	MesP2W   : REAL ; 
	MesP3W   : REAL ; 
	MesQ1W   : REAL ; 
	MesQ2W   : REAL ; 
	MesQ3W   : REAL ; 
	MesQW	 : REAL ; 
	CalSW	: REAL ; 
	
	CalEacdelWh	: REAL ; 
	CalEarecWh	: REAL ; 	
	CalEreacdelvah	: REAL ; 
	CalErearecvah	: REAL ; 

	
END_VAR
//INITIALIZING MODBUS REQUESTS //
	FB_ModbusRead_I1[1](Reset:= CmdClearFault_G ,sIPAddr:=ParamIpAddress, tTimeout:= ParamTimeout,nTcpPort:=502);

// CP-Read / Write 

MesDataExd.MesData.MesCP_Read := MesCP_Read ; 


IF MesCP_Read  THEN	
// MODBUS REQUEST//
	FB_ModbusRead_I1[1](
		nQuantity		:= 122, 
		nMBAddr			:= 19000, 
		nUnitID			:= ParamUnitID,
		cbLength		:= SIZEOF(MesBlock1_Temp) , 
		pDestAddr		:= ADR(MesBlock1_Temp) ,
		ClockRead		:= MesCP_Read AND ClockRead ,
		ModbusReadAlarm	=>	MesModbusReadAlarm[1] , 
		ErrorId			=> MesModbusAlarmCode);

// PROPERTIES UPDATE // 


	// Block 1
MW( WORD_STRONG:= MesBlock1_Temp[26], WORD_WEAK := MesBlock1_Temp[27], VAR_OUT:=MesPW);
MW( WORD_STRONG:= MesBlock1_Temp[42], WORD_WEAK := MesBlock1_Temp[43], VAR_OUT:=MesQW);
MW( WORD_STRONG:= MesBlock1_Temp[44], WORD_WEAK := MesBlock1_Temp[45], VAR_OUT:=MesDataExd.MesData.MesCosPhi1);
MW( WORD_STRONG:= MesBlock1_Temp[46], WORD_WEAK := MesBlock1_Temp[47], VAR_OUT:=MesDataExd.MesData.MesCosPhi2);
MW( WORD_STRONG:= MesBlock1_Temp[48], WORD_WEAK := MesBlock1_Temp[49], VAR_OUT:=MesDataExd.MesData.MesCosPhi3);
MW( WORD_STRONG:= MesBlock1_Temp[0], WORD_WEAK := MesBlock1_Temp[1], VAR_OUT:=MesDataExd.MesData.MesV1);
MW( WORD_STRONG:= MesBlock1_Temp[2], WORD_WEAK := MesBlock1_Temp[3], VAR_OUT:=MesDataExd.MesData.MesV2);
MW( WORD_STRONG:= MesBlock1_Temp[4], WORD_WEAK := MesBlock1_Temp[5], VAR_OUT:=MesDataExd.MesData.MesV3);
MW( WORD_STRONG:= MesBlock1_Temp[6], WORD_WEAK := MesBlock1_Temp[7], VAR_OUT:=MesDataExd.MesData.MesU12);
MW( WORD_STRONG:= MesBlock1_Temp[8], WORD_WEAK := MesBlock1_Temp[9], VAR_OUT:=MesDataExd.MesData.MesU23);
MW( WORD_STRONG:= MesBlock1_Temp[10], WORD_WEAK := MesBlock1_Temp[11], VAR_OUT:=MesDataExd.MesData.MesU31);
MW( WORD_STRONG:= MesBlock1_Temp[12], WORD_WEAK := MesBlock1_Temp[13], VAR_OUT:=MesDataExd.MesData.MesI1);
MW( WORD_STRONG:= MesBlock1_Temp[14], WORD_WEAK := MesBlock1_Temp[15], VAR_OUT:=MesDataExd.MesData.MesI2);
MW( WORD_STRONG:= MesBlock1_Temp[16], WORD_WEAK := MesBlock1_Temp[17], VAR_OUT:=MesDataExd.MesData.MesI3);
MW( WORD_STRONG:= MesBlock1_Temp[50], WORD_WEAK := MesBlock1_Temp[51], VAR_OUT:=MesDataExd.MesData.MesFreq);

MW( WORD_STRONG:= MesBlock1_Temp[20], WORD_WEAK := MesBlock1_Temp[21], VAR_OUT:=MesP1W);
MW( WORD_STRONG:= MesBlock1_Temp[22], WORD_WEAK := MesBlock1_Temp[23], VAR_OUT:=MesP2W);
MW( WORD_STRONG:= MesBlock1_Temp[24], WORD_WEAK := MesBlock1_Temp[25], VAR_OUT:=MesP3W);
MW( WORD_STRONG:= MesBlock1_Temp[36], WORD_WEAK := MesBlock1_Temp[37], VAR_OUT:=MesQ1W);
MW( WORD_STRONG:= MesBlock1_Temp[38], WORD_WEAK := MesBlock1_Temp[39], VAR_OUT:=MesQ2W);
MW( WORD_STRONG:= MesBlock1_Temp[40], WORD_WEAK := MesBlock1_Temp[41], VAR_OUT:=MesQ3W);
MW( WORD_STRONG:= MesBlock1_Temp[34], WORD_WEAK := MesBlock1_Temp[35], VAR_OUT:=CalSW);


MW( WORD_STRONG:= MesBlock1_Temp[68], WORD_WEAK := MesBlock1_Temp[69], VAR_OUT:=CalEarecWh);
MW( WORD_STRONG:= MesBlock1_Temp[76], WORD_WEAK := MesBlock1_Temp[74], VAR_OUT:=CalEacdelWh);
MW( WORD_STRONG:= MesBlock1_Temp[100], WORD_WEAK := MesBlock1_Temp[101], VAR_OUT:=CalErearecvah);
MW( WORD_STRONG:= MesBlock1_Temp[108], WORD_WEAK := MesBlock1_Temp[109], VAR_OUT:=CalEreacdelvah);




// Properties Update 	
MesDataExd.MesData.MesP		:= MesPW / 1000 ; // kW 
MesDataExd.MesData.MesP1		:= MesP1W / 1000 ; 
MesDataExd.MesData.MesP2       := MesP2W / 1000 ; 
MesDataExd.MesData.MesP3       := MesP3W / 1000 ; 
MesDataExd.MesData.MesQ        := MesQW / 1000 ; 
MesDataExd.MesData.MesQ1       := MesQ1W / 1000 ; 
MesDataExd.MesData.MesQ2       := MesQ2W / 1000 ; 
MesDataExd.MesData.MesQ3       := MesQ3W / 1000 ; 
MesDataExd.MesData.MesS		:= CalSW / 1000 ; 

MesDataExd.MesData.MesEActProd		:= CalEacdelWh /1000 ; // kWh 
MesDataExd.MesData.MesEActCons		:= CalEarecWh / 1000 ; 
MesDataExd.MesData.MesEReactProd	:= CalEreacdelvah /1000 ; 
MesDataExd.MesData.MesEReactCons	:= CalErearecvah / 1000  ; 
END_IF 

MesDataExd.MesData.MesCosPhi    := (MesDataExd.MesData.MesCosPhi1 + MesDataExd.MesData.MesCosPhi2 + MesDataExd.MesData.MesCosPhi3)/3;
MesDataExd.MesData.MesI 		:= (MesDataExd.MesData.MesI1 + MesDataExd.MesData.MesI2 + MesDataExd.MesData.MesI3 )/3 ; 
MesDataExd.MesData.MesU			:= (MesDataExd.MesData.MesU12 + MesDataExd.MesData.MesU23 + MesDataExd.MesData.MesU31 ) /3 ; 
MesDataExd.MesData.MesV			:= (MesDataExd.MesData.MesV1 + MesDataExd.MesData.MesV2 + MesDataExd.MesData.MesV3 ) /3 ;

MesDataExd.MesData.MesCosPhi     := (MesDataExd.MesData.MesCosPhi1 + MesDataExd.MesData.MesCosPhi2 + MesDataExd.MesData.MesCosPhi3)/3;
MesDataExd.MesData.MesI :=  ( MesDataExd.MesData.MesI1 + MesDataExd.MesData.MesI2 + MesDataExd.MesData.MesI3 )/3 ; 
MesDataExd.MesData.MesU		:= 	(MesDataExd.MesData.MesU12 + MesDataExd.MesData.MesU23 + MesDataExd.MesData.MesU31 ) /3 ; 
MesDataExd.MesData.MesV		:= 	(MesDataExd.MesData.MesV1 + MesDataExd.MesData.MesV2 + MesDataExd.MesData.MesV3 ) /3 ; 

IF MesDataExd.MesData.MesP > 0.01 OR MesDataExd.MesData.MesP < -0.01 THEN
MesDataExd.MesData.MesTanPhi := MesDataExd.MesData.MesQ /MesDataExd.MesData.MesP;
ELSE
MesDataExd.MesData.MesTanPhi := 0;
END_IF
END_METHOD

END_FUNCTION_BLOCK

// ---- 01_Equipement_Library/Operation Meter/FB_PM_PM800.TcPOU
FUNCTION_BLOCK FB_PM_PM800 EXTENDS FB_PM_Base
VAR_INPUT
	{attribute 'OPC.UA.DA' := '1'} 
	ParamIPAddress 	: STRING;	(* (NA) IP Adress of PM 800.*)
END_VAR
VAR_OUTPUT
END_VAR
VAR
MesDataExd AT %Q*	: PM_PM800 ;
	
	// Modbus Read Variables
	FB_ModbusReadAI : ARRAY[1..2] OF FB_ModbusRead ;
	
	// Temp Blocks Filled by Requests
	AI_List_1 	    : ARRAY[1..128] OF WORD ;
	AI_List_2 		: ARRAY[1..128] OF WORD ;
	
	tTimeout 		: TIME := T#2S ;
	
END_VAR

METHOD M_AlarmManagement
VAR_INPUT
END_VAR
//////////////////
// Digiware measurement tool alarm and warning management
/////////////////

VAR 
	// Method local variables (reinitialized at each cycle) 
	FB_AlarmCodeManager			: FB_AlarmCodeManager ; 
	
	ComWarning					: BOOL;			// Error in one of the Modbus Requests
	ComAlarm					: BOOL;			// Error in both Modbus Requests
	
END_VAR
ComWarning 	:= FB_ModbusReadAI[1].ModbusReadAlarm OR FB_ModbusReadAI[2].ModbusReadAlarm;
ComAlarm 	:= FB_ModbusReadAI[1].ModbusReadAlarm AND FB_ModbusReadAI[2].ModbusReadAlarm;
	
TON_ComAlarm(IN:= ComAlarm , PT:= ParamTempoComAlarm, Q= MesDataExd.MesData.MesAlarmCom) ;	
TON_ComWarning(IN:= ComWarning  , PT:= ParamTempoComAlarm, Q=>MesWarningCom) ;	

//					General com alarm : All the read FB fucked up


// ALARM CODE //
	FB_AlarmCodeManager(
		bAlarm1			:= MesDataExd.MesData.MesAlarmCom  , 					// Communication Alarm #COM
		bAlarm2			:=FALSE, // 
		bAlarm3			:=FALSE, // 
		bAlarm4			:=FALSE, // 
		bAlarm5			:=FALSE, //
		bAlarm6			:=FALSE, //
		bAlarm7			:=FALSE, //
		bAlarm8			:=FALSE, //
		bAlarm9			:=FALSE, //
		bAlarm10		:=FALSE, //
		bAlarm11		:=FALSE, //
		bAlarm12		:=FALSE, //
		bAlarm13		:=FALSE, //
		bAlarm14		:=FALSE, //
		bAlarm15		:= FALSE , 			// 			 
		wAlarmCode		=>MesDataExd.MesData.MesAlarmCode);

// WARNING CODE //
	FB_AlarmCodeManager(		
		bAlarm1			:=MesWarningCom	,				 // Communication Warning #COM
		bAlarm2			:=FALSE, 		// 
		bAlarm3			:=FALSE, 		// 
		bAlarm4			:=FALSE, 		// 
		bAlarm5			:=FALSE, //
		bAlarm6			:=FALSE, //
		bAlarm7			:=FALSE, //
		bAlarm8			:=FALSE, //
		bAlarm9			:=FALSE, //
		bAlarm10		:=FALSE, //
		bAlarm11		:=FALSE, //
		bAlarm12		:=FALSE, //
		bAlarm13		:=FALSE, //
		bAlarm14		:=FALSE, //
		bAlarm15		:=FALSE, //
		wAlarmCode		=>MesDataExd.MesData.MesWarningCode);		

// EVENT CODE //
END_METHOD

METHOD M_Read
VAR_INPUT
END_VAR
VAR
	MW					: FB_MergeWordsToDint;
	Test : REAL;
END_VAR
// CP-Read / Write 

MesDataExd.MesData.MesCP_Read := MesCP_Read ; 


IF MesCP_Read  THEN	

// Analogic Inputs Modbus Requests

FB_ModbusReadAI[1](pDestAddr := ADR(AI_List_1),
				sIPAddr := ParamIPAddress,
				tTimeout := tTimeout,
				nTcpPort := 502,
				nQuantity := 110,
				nMBAddr := 1099,
				cbLength := SIZEOF(AI_List_1),
				nUnitID := 1,
				ClockRead := MesCP_Read AND ClockRead,
				Reset := CmdClearFault_G OR IN_CmdReset_L);
				
FB_ModbusReadAI[2](pDestAddr := ADR(AI_List_2),
				sIPAddr := ParamIPAddress,
				tTimeout := tTimeout,
				nTcpPort := 502,
				nQuantity := 18,
				nMBAddr := 1699,
				cbLength := SIZEOF(AI_List_2),
				nUnitID := 1,
				ClockRead := MesCP_Read AND ClockRead,
				Reset := CmdClearFault_G OR IN_CmdReset_L);
				
//  MesDataExd.MesData.Filling Analogic Data			           
				                                
MW(WORD_STRONG :=  AI_List_1[1  ],	WORD_WEAK := AI_List_1[1  ], SIZE := 1, FIX := 0, SIGNED := 0, VAR_OUT	:= MesDataExd.MesData.MesI1);
MW(WORD_STRONG :=  AI_List_1[2  ],	WORD_WEAK := AI_List_1[2  ], SIZE := 1, FIX := 0, SIGNED := 0, VAR_OUT	:= MesDataExd.MesData.MesI2);
MW(WORD_STRONG :=  AI_List_1[3  ],	WORD_WEAK := AI_List_1[3  ], SIZE := 1, FIX := 0, SIGNED := 0, VAR_OUT	:= MesDataExd.MesData.MesI3);
MW(WORD_STRONG :=  AI_List_1[6  ],	WORD_WEAK := AI_List_1[6  ], SIZE := 1, FIX := 0, SIGNED := 0, VAR_OUT	:= MesDataExd.MesData.MesI);
MW(WORD_STRONG :=  AI_List_1[21 ],	WORD_WEAK := AI_List_1[21 ], SIZE := 1, FIX := 0, SIGNED := 0, VAR_OUT	:= MesDataExd.MesData.MesU12);
MW(WORD_STRONG :=  AI_List_1[22 ],	WORD_WEAK := AI_List_1[22 ], SIZE := 1, FIX := 0, SIGNED := 0, VAR_OUT	:= MesDataExd.MesData.MesU23);
MW(WORD_STRONG :=  AI_List_1[23 ],	WORD_WEAK := AI_List_1[23 ], SIZE := 1, FIX := 0, SIGNED := 0, VAR_OUT	:= MesDataExd.MesData.MesU31);
MW(WORD_STRONG :=  AI_List_1[44 ],	WORD_WEAK := AI_List_1[44 ], SIZE := 1, FIX := 0, SIGNED := 0, VAR_OUT	:= MesDataExd.MesData.MesP);
MW(WORD_STRONG :=  AI_List_1[48 ],	WORD_WEAK := AI_List_1[48 ], SIZE := 1, FIX := 0, SIGNED := 0, VAR_OUT	:= MesDataExd.MesData.MesQ);
MW(WORD_STRONG :=  AI_List_1[64 ],	WORD_WEAK := AI_List_1[64 ], SIZE := 1, FIX := 3, SIGNED := 0, VAR_OUT	:= MesDataExd.MesData.MesCosPhi);
MW(WORD_STRONG :=  AI_List_1[81 ],	WORD_WEAK := AI_List_1[81 ], SIZE := 1, FIX := 0, SIGNED := 0, VAR_OUT	:= MesDataExd.MesData.MesFreq);

MW(WORD_STRONG :=  AI_List_1[101],	WORD_WEAK := AI_List_1[101], SIZE := 1, FIX := 0, SIGNED := 0, VAR_OUT	:= MesDataExd.MesTHD1);
MW(WORD_STRONG :=  AI_List_1[102],	WORD_WEAK := AI_List_1[102], SIZE := 1, FIX := 0, SIGNED := 0, VAR_OUT	:= MesDataExd.MesTHD2);
MW(WORD_STRONG :=  AI_List_1[103],	WORD_WEAK := AI_List_1[103], SIZE := 1, FIX := 0, SIGNED := 0, VAR_OUT	:= MesDataExd.MesTHD3);
MW(WORD_STRONG :=  AI_List_1[108],	WORD_WEAK := AI_List_1[108], SIZE := 1, FIX := 0, SIGNED := 0, VAR_OUT	:= MesDataExd.MesTHD1N);
MW(WORD_STRONG :=  AI_List_1[109],	WORD_WEAK := AI_List_1[109], SIZE := 1, FIX := 0, SIGNED := 0, VAR_OUT	:= MesDataExd.MesTHD2N);
MW(WORD_STRONG :=  AI_List_1[110],	WORD_WEAK := AI_List_1[110], SIZE := 1, FIX := 0, SIGNED := 0, VAR_OUT	:= MesDataExd.MesTHD3N);

MesDataExd.MesData.MesEActProd 	:= (WORD_TO_REAL(AI_List_2[1  ]) + WORD_TO_REAL(AI_List_2[2  ])*10000 + WORD_TO_REAL(AI_List_2[3  ])*100000000 + WORD_TO_REAL(AI_List_2[4  ])*1000000000000)/1000;
MesDataExd.MesData.MesEReactProd := (WORD_TO_REAL(AI_List_2[5  ]) + WORD_TO_REAL(AI_List_2[6  ])*10000 + WORD_TO_REAL(AI_List_2[7  ])*100000000 + WORD_TO_REAL(AI_List_2[8  ])*1000000000000)/1000;
MesDataExd.MesData.MesEActCons 	:= (WORD_TO_REAL(AI_List_2[9  ]) + WORD_TO_REAL(AI_List_2[10 ])*10000 + WORD_TO_REAL(AI_List_2[11 ])*100000000 + WORD_TO_REAL(AI_List_2[12  ])*1000000000000)/1000;
MesDataExd.MesData.MesEReactCons := (WORD_TO_REAL(AI_List_2[13 ]) + WORD_TO_REAL(AI_List_2[14 ])*10000 + WORD_TO_REAL(AI_List_2[15 ])*100000000 + WORD_TO_REAL(AI_List_2[16  ])*1000000000000)/1000;	


END_IF
END_METHOD

END_FUNCTION_BLOCK

// ---- 01_Equipement_Library/Operation Meter/FB_PM_Q100.TcPOU
FUNCTION_BLOCK FB_PM_Q100 EXTENDS FB_PM_Base
VAR_INPUT
		ParamIPAddress				: STRING 	:= '192.168.20.66'; 	(* (NA)Config: IP Adress of PV INverter	*)
		ParamUnitID 				: BYTE  	:= 1; 			  		(* (NA)   Modbus Unit ID.               *)
		ParamTCPPort				: UINT		:= 502;					(* (NA) TCP port for modbus             *)

END_VAR
VAR_OUTPUT
END_VAR
VAR
	// M_READ VARIABLES//
	MesDataExd			: PM_Q100;
		AX_SB						: ARRAY [1..CstNbSB] OF SB;
		AX_ModbusRead		   		: ARRAY [1..3] OF FB_ModbusRead ; 					// (NA) FB for Modbus Reading
		
		MesBlock1_Temp 				: ARRAY[1..2]  OF WORD; 			// (NA) Temporary Block with multiple modbus reading (Caution : Double Word variables)
		MesBlock2_Temp 				: ARRAY[1..76]  OF WORD; 			// (NA) Temporary Block with multiple modbus reading (Caution : Double Word variables)
		MesBlock3_Temp 				: ARRAY[1..38]  OF WORD; 			// (NA) Temporary Block with multiple modbus reading (Caution : Double Word variables)

		AX_ReadAlarm 		  		: ARRAY [1..3] OF BOOL ; 							// (NA) Modbus Read Alarm for all modbus frames		
		AX_ReadAlarmCode			: ARRAY [1..3] OF UDINT;							// (NA) Modbus Read Alarm Code		
		AX_ReadBusy					: ARRAY [1..3] OF BOOL;								// (NA) Modbus Read Busy  
		AX_ReadCompleted			: ARRAY [1..3] OF BOOL;								// (NA) Modbus Read Completed
				
	

END_VAR

METHOD M_AlarmManagement
//////////////////
// Manages IntelliGen Alarms
/////////////////

VAR 
	// Method local variables (reinitialized at each cycle) 
	FB_AlarmCodeManager : FB_AlarmCodeManager ; 

	KK					: BYTE;		// For Loop 
	
	ComWarning			: BOOL;		// Aggregated Wcommunication warning
	ComAlarm			: BOOL;		// Aggregated communication Alarm

END_VAR
	//Alarm
	TON_ComAlarm(IN:= (AX_ModbusRead[1].ModbusReadAlarm) AND (AX_ModbusRead[2].ModbusReadAlarm) AND (AX_ModbusRead[3].ModbusReadAlarm) , PT:= ParamTempoComAlarm, Q= MesDataExd.MesData.MesComAlarm) ;	

	// Alarms if ALL MODBUS frames didn't work and timeout of 15s
	
	
// ALARM CODE //
	FB_AlarmCodeManager(
		bAlarm1			:= MesDataExd.MesData.MesComAlarm,			// Communication general alarm (desactivate if LOC) 
		bAlarm2			:= FALSE,						//
		bAlarm3			:= FALSE, 						//
		bAlarm4			:= FALSE, 		            	//  
		bAlarm5			:= FALSE, 						//
		bAlarm6			:= FALSE, 						//
		bAlarm7			:= False, 						//
		bAlarm8			:= False, 						//
		bAlarm9			:= FALSE, 						//
		bAlarm10		:= FALSE, 						//
		bAlarm11		:= FALSE,                       //
		bAlarm12		:= FALSE,                       //
		bAlarm13		:= FALSE,                       //
		bAlarm14		:= FALSE, 						//
		bAlarm15		:= FALSE, 		                //
		wAlarmCode		=>MesDataExd.MesData.MesAlarmCode);
END_METHOD

METHOD M_CP
//////////////////
//  Emulator
/////////////////

VAR 
	// Method local variables (reinitialized at each cycle) 
	
END_VAR
Trig_Cmd_Read(CLK:=IN_CmdToggleRead);

IF Trig_Cmd_Read.Q THEN
	//IN_CmdToggleRead := FALSE;
MesDataExd.MesData.MesCP_Read := NOT MesDataExd.MesData.MesCP_Read;
END_IF
END_METHOD

METHOD M_Execute
//////////////////
//  Method Calls 
/////////////////

VAR 
	// Method local variables (reinitialized at each cycle) 

END_VAR
IF NOT bInit THEN
	M_Init();
END_IF


SUPER^.M_Execute() ;
END_METHOD

METHOD M_Read
//////////////////
//  Read Modbus Variable for PCS . 
/////////////////
VAR 
	// Method local variables (reinitialized at each cycle) 
		MW 					: FB_MergeWordsToFloat; 
		MW1					: FB_MergeWordsToDint;
		
	KK: INT;
	MesWarningCodeAkuo: INT;
	MesPTemp: REAL;
	MesQTemp: REAL;
END_VAR
// CP-Read / Write 

MesDataExd.MesData.MesCP_Read := MesCP_Read ; 
 

IF MesCP_Read  THEN		
	
	AX_ModbusRead[1]
	(
		pDestAddr := ADR(MesBlock1_Temp),
		sIPAddr := ParamIPAddress,
		tTimeout := ParamTimeout,
		nQuantity := 2,
		ntcpport := ParamTCPPort,
		nMBAddr := 100,
		nUnitID := ParamUnitID,
		cbLength := SIZEOF(MesBlock1_Temp),
		ClockRead := ClockRead,
		Reset := CmdClearFault_G OR IN_CmdReset_L,
		ErrorId => AX_ReadAlarmCode[1],
		ModbusReadAlarm => AX_ReadAlarm[1],
		Busy => AX_ReadBusy[1]	
	);
	
	AX_ModbusRead[2]
	(
		pDestAddr := ADR(MesBlock2_Temp),
		sIPAddr := ParamIPAddress,
		tTimeout := ParamTimeout,
		nQuantity := 76,
		ntcpport := ParamTCPPort,
		nMBAddr := 200,
		nUnitID := ParamUnitID,
		cbLength := SIZEOF(MesBlock2_Temp),
		ClockRead := ClockRead,
		Reset := CmdClearFault_G OR IN_CmdReset_L,
		ErrorId => AX_ReadAlarmCode[2],
		ModbusReadAlarm => AX_ReadAlarm[2],
		Busy => AX_ReadBusy[2]	
	);
	
	AX_ModbusRead[3]
	(
		pDestAddr := ADR(MesBlock3_Temp),
		sIPAddr := ParamIPAddress,
		tTimeout := ParamTimeout,
		nQuantity := 38,
		ntcpport := ParamTCPPort,
		nMBAddr := 800,
		nUnitID := ParamUnitID,
		cbLength := SIZEOF(MesBlock3_Temp),
		ClockRead := ClockRead,
		Reset := CmdClearFault_G OR IN_CmdReset_L,
		ErrorId => AX_ReadAlarmCode[3],
		ModbusReadAlarm => AX_ReadAlarm[3],
		Busy => AX_ReadBusy[3]	
	);
	
	FOR KK := 1 TO 3 DO
		AX_ReadCompleted[KK] := NOT AX_ReadAlarm[KK] AND NOT AX_ReadBusy[KK];
	END_FOR
	
MesDataExd.MesState1 := MesBlock1_Temp[1];
MesDataExd.MesState2 := MesBlock1_Temp[2];
	
	MW( WORD_STRONG:= MesBlock2_Temp[ 1], 	WORD_WEAK := MesBlock2_Temp[ 2],	VAR_OUT := MesDataExd.MesData.MesV1);
	MW( WORD_STRONG:= MesBlock2_Temp[ 3], 	WORD_WEAK := MesBlock2_Temp[ 4],	VAR_OUT := MesDataExd.MesData.MesV2);
	MW( WORD_STRONG:= MesBlock2_Temp[ 5], 	WORD_WEAK := MesBlock2_Temp[ 6],	VAR_OUT := MesDataExd.MesData.MesV3);
	MW( WORD_STRONG:= MesBlock2_Temp[ 7], 	WORD_WEAK := MesBlock2_Temp[ 8],	VAR_OUT := MesDataExd.MesVN);
	MW( WORD_STRONG:= MesBlock2_Temp[ 9], 	WORD_WEAK := MesBlock2_Temp[10],	VAR_OUT := MesDataExd.MesData.MesI1);
	MW( WORD_STRONG:= MesBlock2_Temp[11], 	WORD_WEAK := MesBlock2_Temp[12],	VAR_OUT := MesDataExd.MesData.MesI2);
	MW( WORD_STRONG:= MesBlock2_Temp[13], 	WORD_WEAK := MesBlock2_Temp[14],	VAR_OUT := MesDataExd.MesData.MesI3);
	MW( WORD_STRONG:= MesBlock2_Temp[15], 	WORD_WEAK := MesBlock2_Temp[16],	VAR_OUT := MesDataExd.MesData.MesIN);
	MW( WORD_STRONG:= MesBlock2_Temp[17], 	WORD_WEAK := MesBlock2_Temp[18], 	VAR_OUT := MesDataExd.MesData.MesU12);
	MW( WORD_STRONG:= MesBlock2_Temp[19], 	WORD_WEAK := MesBlock2_Temp[20], 	VAR_OUT := MesDataExd.MesData.MesU23);
	MW( WORD_STRONG:= MesBlock2_Temp[21], 	WORD_WEAK := MesBlock2_Temp[22], 	VAR_OUT := MesDataExd.MesData.MesU31);
	MW( WORD_STRONG:= MesBlock2_Temp[23], 	WORD_WEAK := MesBlock2_Temp[24],  VAR_OUT := MesDataExd.MesData.MesV);
	MW( WORD_STRONG:= MesBlock2_Temp[25], 	WORD_WEAK := MesBlock2_Temp[26],  VAR_OUT := MesDataExd.MesData.MesI);
	MW( WORD_STRONG:= MesBlock2_Temp[27], 	WORD_WEAK := MesBlock2_Temp[28],  VAR_OUT := MesDataExd.MesData.MesP1);
	MW( WORD_STRONG:= MesBlock2_Temp[29], 	WORD_WEAK := MesBlock2_Temp[30],  VAR_OUT := MesDataExd.MesData.MesP2);
	MW( WORD_STRONG:= MesBlock2_Temp[31], 	WORD_WEAK := MesBlock2_Temp[32],  VAR_OUT := MesDataExd.MesData.MesP3);
	MW( WORD_STRONG:= MesBlock2_Temp[33], 	WORD_WEAK := MesBlock2_Temp[34],  VAR_OUT := MesPTemp);
	MW( WORD_STRONG:= MesBlock2_Temp[35], 	WORD_WEAK := MesBlock2_Temp[36],  VAR_OUT := MesDataExd.MesData.MesQ1);
	MW( WORD_STRONG:= MesBlock2_Temp[37], 	WORD_WEAK := MesBlock2_Temp[38],  VAR_OUT := MesDataExd.MesData.MesQ2);
	MW( WORD_STRONG:= MesBlock2_Temp[39], 	WORD_WEAK := MesBlock2_Temp[40],  VAR_OUT := MesDataExd.MesData.MesQ3);
	MW( WORD_STRONG:= MesBlock2_Temp[41], 	WORD_WEAK := MesBlock2_Temp[42],  VAR_OUT := MesQTemp);
	MW( WORD_STRONG:= MesBlock2_Temp[43], 	WORD_WEAK := MesBlock2_Temp[44],  VAR_OUT := MesDataExd.MesData.MesS1);
	MW( WORD_STRONG:= MesBlock2_Temp[45], 	WORD_WEAK := MesBlock2_Temp[46],  VAR_OUT := MesDataExd.MesData.MesS2);
	MW( WORD_STRONG:= MesBlock2_Temp[47], 	WORD_WEAK := MesBlock2_Temp[48],  VAR_OUT := MesDataExd.MesData.MesS3);
	MW( WORD_STRONG:= MesBlock2_Temp[49], 	WORD_WEAK := MesBlock2_Temp[50],  VAR_OUT := MesDataExd.MesData.MesS);
	MW( WORD_STRONG:= MesBlock2_Temp[75], 	WORD_WEAK:= MesBlock2_Temp[76], VAR_OUT:= MesDataExd.MesData.MesFreq);
																			
																			
	MW( WORD_STRONG:= MesBlock3_Temp[01], 	WORD_WEAK := MesBlock3_Temp[02], VAR_OUT:= MesDataExd.MesEPerPulse);
	MW1( WORD_STRONG:= MesBlock3_Temp[07], 	WORD_WEAK := MesBlock3_Temp[08], Size := 2, fix := 0, signed := FALSE, VAR_OUT := MesDataExd.MesEac1_dmd);
	MW1( WORD_STRONG:= MesBlock3_Temp[09], 	WORD_WEAK := MesBlock3_Temp[10], Size := 2, fix := 0, signed := FALSE, VAR_OUT := MesDataExd.MesEac2_dmd);
	MW1( WORD_STRONG:= MesBlock3_Temp[11], 	WORD_WEAK := MesBlock3_Temp[12], Size := 2, fix := 0, signed := FALSE, VAR_OUT := MesDataExd.MesEac3_dmd);
	MW1( WORD_STRONG:= MesBlock3_Temp[13], 	WORD_WEAK := MesBlock3_Temp[14], Size := 2, fix := 0, signed := FALSE, VAR_OUT := MesDataExd.MesEac_dmd );
	MW1( WORD_STRONG:= MesBlock3_Temp[15], 	WORD_WEAK := MesBlock3_Temp[16], Size := 2, fix := 0, signed := FALSE, VAR_OUT := MesDataExd.MesEac1_sup);
	MW1( WORD_STRONG:= MesBlock3_Temp[17], 	WORD_WEAK := MesBlock3_Temp[18], Size := 2, fix := 0, signed := FALSE, VAR_OUT := MesDataExd.MesEac2_sup);
	MW1( WORD_STRONG:= MesBlock3_Temp[19], 	WORD_WEAK := MesBlock3_Temp[20], Size := 2, fix := 0, signed := FALSE, VAR_OUT := MesDataExd.MesEac3_sup);
	MW1( WORD_STRONG:= MesBlock3_Temp[21], 	WORD_WEAK := MesBlock3_Temp[22], Size := 2, fix := 0, signed := FALSE, VAR_OUT := MesDataExd.MesEac_sup );
	MW1( WORD_STRONG:= MesBlock3_Temp[23], 	WORD_WEAK := MesBlock3_Temp[24], Size := 2, fix := 0, signed := FALSE, VAR_OUT := MesDataExd.MesEreac1_ind);
	MW1( WORD_STRONG:= MesBlock3_Temp[25], 	WORD_WEAK := MesBlock3_Temp[26], Size := 2, fix := 0, signed := FALSE, VAR_OUT := MesDataExd.MesEreac2_ind);
	MW1( WORD_STRONG:= MesBlock3_Temp[27], 	WORD_WEAK := MesBlock3_Temp[28], Size := 2, fix := 0, signed := FALSE, VAR_OUT := MesDataExd.MesEreac3_ind);
	MW1( WORD_STRONG:= MesBlock3_Temp[29], 	WORD_WEAK := MesBlock3_Temp[30], Size := 2, fix := 0, signed := FALSE, VAR_OUT := MesDataExd.MesEreac_ind );
	MW1( WORD_STRONG:= MesBlock3_Temp[31], 	WORD_WEAK := MesBlock3_Temp[32], Size := 2, fix := 0, signed := FALSE, VAR_OUT := MesDataExd.MesEreac1_cap);
	MW1( WORD_STRONG:= MesBlock3_Temp[33], 	WORD_WEAK := MesBlock3_Temp[34], Size := 2, fix := 0, signed := FALSE, VAR_OUT := MesDataExd.MesEreac2_cap);
	MW1( WORD_STRONG:= MesBlock3_Temp[35], 	WORD_WEAK := MesBlock3_Temp[36], Size := 2, fix := 0, signed := FALSE, VAR_OUT := MesDataExd.MesEreac3_cap);
	MW1( WORD_STRONG:= MesBlock3_Temp[37], 	WORD_WEAK := MesBlock3_Temp[38], Size := 2, fix := 0, signed := FALSE, VAR_OUT := MesDataExd.MesEreac_cap);
	
MesDataExd.CalEac1_dmd      := MesDataExd.MesEac1_dmd        * MesDataExd.MesEPerPulse ;
MesDataExd.CalEac2_dmd      := MesDataExd.MesEac2_dmd        * MesDataExd.mesEperpulse ;
MesDataExd.CalEac3_dmd      := MesDataExd.MesEac3_dmd        * MesDataExd.mesEperpulse ;
MesDataExd.CalEac_dmd       := MesDataExd.MesEac_dmd         * MesDataExd.mesEperpulse ;
MesDataExd.CalEac1_sup      := MesDataExd.MesEac1_sup        * MesDataExd.mesEperpulse ;
MesDataExd.CalEac2_sup      := MesDataExd.MesEac2_sup        * MesDataExd.mesEperpulse ;
MesDataExd.CalEac3_sup      := MesDataExd.MesEac3_sup        * MesDataExd.mesEperpulse ;
MesDataExd.CalEac_sup       := MesDataExd.MesEac_sup         * MesDataExd.mesEperpulse ;
MesDataExd.CalEreac1_ind    := MesDataExd.MesEreac1_ind      * MesDataExd.mesEperpulse ;
MesDataExd.CalEreac2_ind    := MesDataExd.MesEreac2_ind      * MesDataExd.mesEperpulse ;
MesDataExd.CalEreac3_ind    := MesDataExd.MesEreac3_ind      * MesDataExd.mesEperpulse ;
MesDataExd.CalEreac_ind     := MesDataExd.MesEreac_ind       * MesDataExd.mesEperpulse ;
MesDataExd.CalEreac1_cap    := MesDataExd.MesEreac1_cap      * MesDataExd.mesEperpulse ;
MesDataExd.CalEreac2_cap    := MesDataExd.MesEreac2_cap      * MesDataExd.mesEperpulse ;
MesDataExd.CalEreac3_cap    := MesDataExd.MesEreac3_cap      * MesDataExd.mesEperpulse ;
MesDataExd.CalEreac_cap     := MesDataExd.MesEreac_cap       * MesDataExd.mesEperpulse ;
	
	// Changement signe P 
	
MesDataExd.MesData.MesP := -MesPTemp/1000;
MesDataExd.MesData.MesQ := -MesQTemp/1000;
MesDataExd.MesData.MesU := SQRT(3)*MesDataExd.MesData.MesV;
	
	IF ABS(MesDataExd.MesData.MesP) > 0 THEN
	MesDataExd.MesData.MesTanPhi := MesDataExd.MesData.MesQ / ABS(MesDataExd.MesData.MesP);
	END_IF


END_IF
END_METHOD

END_FUNCTION_BLOCK

// ---- 01_Equipement_Library/Operation Meter/FB_PM_SM103E.TcPOU
FUNCTION_BLOCK FB_PM_SM103E EXTENDS FB_PM_Base
//////////////////
// Measurement Solution based on Digiware, but access through PMS Socomec
//////////////////
VAR CONSTANT
	// Characteristics of the object (Same for all instances)
			
END_VAR

VAR_INPUT PERSISTENT
	// Parameters of the Object (instance specific) 
	{attribute 'OPC.UA.DA' := '1'} 
	ParamUnitID					: BYTE 		:= 5 ;								// (NA)unit ID
	

END_VAR

VAR_OUTPUT
	//Child objects
	
END_VAR
VAR
	//M_ALARMMANAGEMENT VARIABLES//	                                                    							                                                								

	//M_READ VARIABLES//

	bReadError					: BOOL;
	bReadCompleted 				: BOOL;
	bReadBusy					: BOOL;
	InputStructRead 			: Struct_InputRTU;



	bReadError2					: BOOL;
	bReadCompleted2 				: BOOL;
	bReadBusy2					: BOOL;
	InputStructRead2 			: Struct_InputRTU;
	
	MesBlock1_Temp 				: ARRAY[1..64]  OF WORD; 		// (NA) Temporary Block with multiple mod
	MesBlock2_Temp 				: ARRAY[1..20]  OF WORD; 		// (NA) Temporary Block with multiple mod

		
		
	//M_INIT VARIABLES //
	
	// M_EXECUTE VARIABLES //
		RTrigI						: R_TRIG;

	MesDataExd AT %Q*			: PM_Standard ;

 
END_VAR

METHOD M_AlarmManagement
//////////////////
// Digiware measurement tool alarm and warning management
/////////////////

VAR 
	// Method local variables (reinitialized at each cycle) 
	FB_AlarmCodeManager			: FB_AlarmCodeManager ; 
	
	KK							: BYTE ;		// For loop
	
	CMWarning					: BOOL;			// At least one Digiware device in Alarm
	CMAlarm						: BOOL;			// At least one Digiware device in Alarm
	
END_VAR

CMAlarm := bReadError AND bReadError2 ; 
MesWarningCom := bReadError OR bReadError2 ;

//					General com alarm : All the read FB fucked up
TON_ComAlarm(IN:= CMAlarm , PT:= ParamTempoComAlarm, Q=>MesDataExd.MesData.MesAlarmCom) ;	 	// D50 LOC
// ALARM CODE //
	FB_AlarmCodeManager(
		bAlarm1			:= MesDataExd.MesData.MesAlarmCom   , 					// Communication Error  #COM
		bAlarm2			:=FALSE, 		// 
		bAlarm3			:=FALSE, 		// 
		bAlarm4			:=FALSE, 		// 
		bAlarm5			:=FALSE, 
		bAlarm6			:=FALSE, 
		bAlarm7			:=FALSE, 
		bAlarm8			:=FALSE, 
		bAlarm9			:=FALSE, 
		bAlarm10		:=FALSE, 
		bAlarm11		:=FALSE, 
		bAlarm12		:=FALSE, 
		bAlarm13		:=FALSE, 
		bAlarm14		:=FALSE, 
		bAlarm15		:= FALSE , 			// 							 
		wAlarmCode		=>MesDataExd.MesData.MesAlarmCode);

// WARNING CODE //
	FB_AlarmCodeManager(		
		bAlarm1			:=MesWarningCom	,				 // Communication warning #COM
		bAlarm2			:=FALSE, 		// 
		bAlarm3			:=FALSE, 		// 
		bAlarm4			:=FALSE, 		// 
		bAlarm5			:=FALSE, 
		bAlarm6			:=FALSE, 
		bAlarm7			:=FALSE, 
		bAlarm8			:=FALSE, 
		bAlarm9			:=FALSE, 
		bAlarm10		:=FALSE, 
		bAlarm11		:=FALSE, 
		bAlarm12		:=FALSE, 
		bAlarm13		:=FALSE, 
		bAlarm14		:=FALSE, 
		bAlarm15		:=FALSE, 
		wAlarmCode		=>MesDataExd.MesData.MesWarningCode);
END_METHOD

METHOD M_Init
VAR 

END_VAR
END_METHOD

METHOD M_Read
//////////////////
//  Read Modbus Variable for PCS . 
/////////////////
VAR 
	// Method local variables (reinitialized at each cycle) 
	MW 					: FB_MergeWordsToDint; 
						// FOR Loop 


END_VAR
// CP-Read / Write 

MesDataExd.MesData.MesCP_Read := MesCP_Read ; 


IF MesCP_Read  THEN	

(*
//Metrology

InputStructRead.InBuffer := ADR(MesBlock1_Temp);
InputStructRead.InFunction := 3;
InputStructRead.InQuantity := 54;
InputStructRead.InStartAddr := 768;
InputStructRead.InUnitID := ParamUnitID;

InputStructRead.OutBusy := ADR(bReadBusy);
InputStructRead.OutError := ADR(bReadError);
InputStructRead.OutCompleted := ADR(bReadCompleted);


RTrigI(CLK:= ClockRead );

IF RTrigI.Q THEN 
	A1_SUB_MV.ModbusRTU.M_AddAction_FIFO(InStruct:= InputStructRead , InPriority:=1 ) ; 
END_IF

// Properties update
MW(WORD_STRONG:=MesBlock1_Temp[1] , WORD_WEAK:=MesBlock1_Temp[2] , SIZE:=2, FIX :=3 , SIGNED :=FALSE , VAR_OUT := MesDataExd.MesData.MesI1  ); 
MW(WORD_STRONG:=MesBlock1_Temp[3] , WORD_WEAK:=MesBlock1_Temp[4] , SIZE:=2, FIX :=3 , SIGNED :=FALSE , VAR_OUT := MesDataExd.MesData.MesI2  ); 
MW(WORD_STRONG:=MesBlock1_Temp[5] , WORD_WEAK:=MesBlock1_Temp[6] , SIZE:=2, FIX :=3 , SIGNED :=FALSE , VAR_OUT := MesDataExd.MesData.MesI3  ); 
MW(WORD_STRONG:=MesBlock1_Temp[7] , WORD_WEAK:=MesBlock1_Temp[8] , SIZE:=2, FIX :=3 , SIGNED :=FALSE , VAR_OUT := MesDataExd.MesData.MesIN  ); 
MW(WORD_STRONG:=MesBlock1_Temp[9] , WORD_WEAK:=MesBlock1_Temp[10] , SIZE:=2, FIX :=2 , SIGNED :=FALSE , VAR_OUT := MesDataExd.MesData.MesU12  ); 
MW(WORD_STRONG:=MesBlock1_Temp[11] , WORD_WEAK:=MesBlock1_Temp[12] , SIZE:=2, FIX :=2 , SIGNED :=FALSE , VAR_OUT := MesDataExd.MesData.MesU23  ); 
MW(WORD_STRONG:=MesBlock1_Temp[13] , WORD_WEAK:=MesBlock1_Temp[14] , SIZE:=2, FIX :=2 , SIGNED :=FALSE , VAR_OUT := MesDataExd.MesData.MesU31  ); 
MW(WORD_STRONG:=MesBlock1_Temp[15] , WORD_WEAK:=MesBlock1_Temp[16] , SIZE:=2, FIX :=2 , SIGNED :=FALSE , VAR_OUT := MesDataExd.MesData.MesV1  ); 
MW(WORD_STRONG:=MesBlock1_Temp[17] , WORD_WEAK:=MesBlock1_Temp[18] , SIZE:=2, FIX :=2 , SIGNED :=FALSE , VAR_OUT := MesDataExd.MesData.MesV2  ); 
MW(WORD_STRONG:=MesBlock1_Temp[19] , WORD_WEAK:=MesBlock1_Temp[20] , SIZE:=2, FIX :=2 , SIGNED :=FALSE , VAR_OUT := MesDataExd.MesData.MesV3  ); 
MW(WORD_STRONG:=MesBlock1_Temp[21] , WORD_WEAK:=MesBlock1_Temp[22] , SIZE:=2, FIX :=2 , SIGNED :=FALSE , VAR_OUT := MesDataExd.MesData.MesFreq  ); 
MW(WORD_STRONG:=MesBlock1_Temp[23] , WORD_WEAK:=MesBlock1_Temp[24] , SIZE:=2, FIX :=2 , SIGNED :=TRUE , VAR_OUT := MesDataExd.MesData.MesP  ); 
MW(WORD_STRONG:=MesBlock1_Temp[25] , WORD_WEAK:=MesBlock1_Temp[26] , SIZE:=2, FIX :=2 , SIGNED :=TRUE , VAR_OUT := MesDataExd.MesData.MesQ  ); 
MW(WORD_STRONG:=MesBlock1_Temp[27] , WORD_WEAK:=MesBlock1_Temp[28] , SIZE:=2, FIX :=2 , SIGNED :=FALSE , VAR_OUT := MesDataExd.MesData.MesS  ); 
MW(WORD_STRONG:=MesBlock1_Temp[29] , WORD_WEAK:=MesBlock1_Temp[30] , SIZE:=2, FIX :=3 , SIGNED :=TRUE , VAR_OUT := MesDataExd.MesData.MesPF  ); 
MW(WORD_STRONG:=MesBlock1_Temp[31] , WORD_WEAK:=MesBlock1_Temp[32] , SIZE:=2, FIX :=2 , SIGNED :=TRUE , VAR_OUT := MesDataExd.MesData.MesP1  ); 
MW(WORD_STRONG:=MesBlock1_Temp[33] , WORD_WEAK:=MesBlock1_Temp[34] , SIZE:=2, FIX :=2 , SIGNED :=TRUE , VAR_OUT := MesDataExd.MesData.MesP2  ); 
MW(WORD_STRONG:=MesBlock1_Temp[35] , WORD_WEAK:=MesBlock1_Temp[36] , SIZE:=2, FIX :=2 , SIGNED :=TRUE , VAR_OUT := MesDataExd.MesData.MesP3  ); 
MW(WORD_STRONG:=MesBlock1_Temp[37] , WORD_WEAK:=MesBlock1_Temp[38] , SIZE:=2, FIX :=2 , SIGNED :=TRUE , VAR_OUT := MesDataExd.MesData.MesQ1  ); 
MW(WORD_STRONG:=MesBlock1_Temp[39] , WORD_WEAK:=MesBlock1_Temp[40] , SIZE:=2, FIX :=2 , SIGNED :=TRUE , VAR_OUT := MesDataExd.MesData.MesQ2  ); 
MW(WORD_STRONG:=MesBlock1_Temp[41] , WORD_WEAK:=MesBlock1_Temp[42] , SIZE:=2, FIX :=2 , SIGNED :=TRUE , VAR_OUT := MesDataExd.MesData.MesQ3  ); 
MW(WORD_STRONG:=MesBlock1_Temp[43] , WORD_WEAK:=MesBlock1_Temp[44] , SIZE:=2, FIX :=2 , SIGNED :=FALSE , VAR_OUT := MesDataExd.MesData.MesS1  ); 
MW(WORD_STRONG:=MesBlock1_Temp[45] , WORD_WEAK:=MesBlock1_Temp[46] , SIZE:=2, FIX :=2 , SIGNED :=FALSE , VAR_OUT := MesDataExd.MesData.MesS2  ); 
MW(WORD_STRONG:=MesBlock1_Temp[47] , WORD_WEAK:=MesBlock1_Temp[48] , SIZE:=2, FIX :=2 , SIGNED :=FALSE , VAR_OUT := MesDataExd.MesData.MesS3  ); 
MW(WORD_STRONG:=MesBlock1_Temp[49] , WORD_WEAK:=MesBlock1_Temp[50] , SIZE:=2, FIX :=3 , SIGNED :=TRUE , VAR_OUT := MesDataExd.MesData.MesPF1  ); 
MW(WORD_STRONG:=MesBlock1_Temp[51] , WORD_WEAK:=MesBlock1_Temp[52] , SIZE:=2, FIX :=3 , SIGNED :=TRUE , VAR_OUT := MesDataExd.MesData.MesPF2  ); 
MW(WORD_STRONG:=MesBlock1_Temp[53] , WORD_WEAK:=MesBlock1_Temp[54] , SIZE:=2, FIX :=3 , SIGNED :=TRUE , VAR_OUT := MesDataExd.MesData.MesPF3  ); 
 


MesData.MesI := MesDataExd.MesData.MesI1 + MesDataExd.MesData.MesI2 MesDataExd.MesData.MesI3 ) /3 ; 
MesData.MesU := MesDataExd.MesData.MesU12 + MesDataExd.MesData.MesU23 MesDataExd.MesData.MesU31 ) /3 ; 
MesData.MesV := MesDataExd.MesData.MesV1 + MesDataExd.MesData.MesV2 MesDataExd.MesData.MesV3 ) /3 ; 


//Energy
InputStructRead2.InBuffer := ADR(MesBlock2_Temp);
InputStructRead2.InFunction := 3;
InputStructRead2.InQuantity := 10;
InputStructRead2.InStartAddr := 50780;
InputStructRead2.InUnitID := ParamUnitID;

InputStructRead2.OutBusy := ADR(bReadBusy2);
InputStructRead2.OutError := ADR(bReadError2);
InputStructRead2.OutCompleted := ADR(bReadCompleted2);


IF RTrigI.Q THEN 
	A1_SUB_MV.ModbusRTU.M_AddAction_FIFO(InStruct:= InputStructRead2 , InPriority:=1 ) ; 
END_IF

// Properties update
MW(WORD_STRONG:=MesBlock2_Temp[1] , WORD_WEAK:=MesBlock2_Temp[2] , SIZE:=2, FIX :=0 , SIGNED :=FALSE , VAR_OUT := MesDataExd.MesData.MesEActProd  ); 
MW(WORD_STRONG:=MesBlock2_Temp[3] , WORD_WEAK:=MesBlock2_Temp[4] , SIZE:=2, FIX :=0 , SIGNED :=FALSE , VAR_OUT := MesDataExd.MesData.MesEReactProd  ); 

MW(WORD_STRONG:=MesBlock2_Temp[7] , WORD_WEAK:=MesBlock2_Temp[8] , SIZE:=2, FIX :=0 , SIGNED :=FALSE , VAR_OUT := MesDataExd.MesData.MesEActCons  ); 
MW(WORD_STRONG:=MesBlock2_Temp[9] , WORD_WEAK:=MesBlock2_Temp[10] , SIZE:=2, FIX :=0 , SIGNED :=FALSE , VAR_OUT := MesDataExd.MesData.MesEReactCons  ); 


*)

END_IF
END_METHOD

END_FUNCTION_BLOCK

// ---- 01_Equipement_Library/Operation Meter/FB_PM_PM3250.TcPOU
FUNCTION_BLOCK FB_PM_PM3250 EXTENDS FB_PM_Base
//////////////////
// Measurement Solution based on Digiware, but access through PMS Socomec
//////////////////
VAR CONSTANT
	// Characteristics of the object (Same for all instances)
			
END_VAR

VAR_INPUT PERSISTENT
	// Parameters of the Object (instance specific) 
	{attribute 'OPC.UA.DA' := '1'} 
	ParamUnitID					: BYTE 		:= 1 ;								(* (NA)unit ID*)
//	ParamInInterfaceSub			: BOOL := TRUE; 								// (NA) Serial interface RS422/RS485 TYPE (0:EL6021,1:SUB9)			
END_VAR

VAR_OUTPUT
	//Child objects
	
END_VAR
VAR

	//M_READ VARIABLES//
		InputStructRead 			: ARRAY[1..5] OF  Struct_InputRTU;

		AX_Quantity					: ARRAY[1..5] OF WORD;					// (NA) Quantity of blocks to read
		AX_Address					: ARRAY[1..5] OF WORD;					// (NA) Start address of the read
		MesBlock_Temp 				: ARRAY[1..5] OF ARRAY[1..125] OF WORD;	// (NA) Temporary Block with multiple modbus reading (U30 + I35)
		Busy						: BOOL;
		OutErrorMbRead				: ARRAY[1..5] OF BOOL;
	

	//M_INIT VARIABLES //
		OutFBCompleteted			: BOOL;
	// M_EXECUTE VARIABLES //
		RTrigI						: R_TRIG;
		MesDataExd		AT %Q*			: PM_Standard ;
END_VAR

METHOD M_AlarmManagement
//////////////////
// Digiware measurement tool alarm and warning management
/////////////////

VAR 
	// Method local variables (reinitialized at each cycle) 
	FB_AlarmCodeManager			: FB_AlarmCodeManager ; 
	
	KK							: BYTE ;		// For loop
	
	CMWarning					: BOOL;			// At least one Digiware device in Alarm
	CMAlarm						: BOOL;			// At least one Digiware device in Alarm
	
END_VAR

	
TON_ComAlarm(IN:= OutErrorMbRead[1] AND OutErrorMbRead[2] AND OutErrorMbRead[3] AND OutErrorMbRead[4] AND OutErrorMbRead[5] , PT:= ParamTempoComAlarm, Q=> MesDataExd.MesData.MesAlarmCom) ;	
TON_ComWarning(IN:= OutErrorMbRead[1] OR OutErrorMbRead[2] OR OutErrorMbRead[3] OR OutErrorMbRead[4] OR OutErrorMbRead[5] , PT:= ParamTempoComAlarm, Q=>MesWarningCom) ;	

// General com alarm : All the read FB fucked up
// ALARM CODE //
	FB_AlarmCodeManager( 
		bAlarm1			:= MesDataExd.MesData.MesAlarmCom, 					// Communication Error  #COM
		bAlarm2			:=FALSE, 									// 
		bAlarm3			:=FALSE, 									// 
		bAlarm4			:=FALSE, 									// 
		bAlarm5			:=FALSE, 									//
		bAlarm6			:=FALSE, 									//
		bAlarm7			:=FALSE, 									//
		bAlarm8			:=FALSE, 									//
		bAlarm9			:=FALSE, 									//
		bAlarm10		:=FALSE, 									//
		bAlarm11		:=FALSE, 									//
		bAlarm12		:=FALSE, 									//
		bAlarm13		:=FALSE, 									//
		bAlarm14		:=FALSE, 									//
		bAlarm15		:= FALSE , 									//						 
		wAlarmCode		=>MesDataExd.MesData.MesAlarmCode);

// WARNING CODE //
	FB_AlarmCodeManager(		
		bAlarm1			:=	MesWarningCom,				 			// Communication Warning #COM	
		bAlarm2			:=FALSE, 									// 
		bAlarm3			:=FALSE, 									// 
		bAlarm4			:=FALSE, 									// 
		bAlarm5			:=FALSE, 									//
		bAlarm6			:=FALSE, 									//
		bAlarm7			:=FALSE, 									//
		bAlarm8			:=FALSE, 									//
		bAlarm9			:=FALSE, 									//
		bAlarm10		:=FALSE, 									//
		bAlarm11		:=FALSE, 									//
		bAlarm12		:=FALSE, 									//
		bAlarm13		:=FALSE, 									//
		bAlarm14		:=FALSE, 									//
		bAlarm15		:=FALSE, 									//
		wAlarmCode		=>MesDataExd.MesData.MesWarningCode);
END_METHOD

METHOD M_Evaluate : BOOL
VAR_INPUT
END_VAR
END_METHOD

METHOD M_Execute
//////////////////
//  Method Calls 
/////////////////
VAR 
	// Method local variables (reinitialized at each cycle) 
	// EMULATOR
		Psoltot		: REAL;		// Total Solar Power . 
		KK			: BYTE;		// For Loop
	
END_VAR
// READING AND WRITING CLOCK //
	TP1(IN:=NOT TP1.Q , PT:= ParamClockReadTime);
	ClockRead 		:= TP1.Q;

// PERMANENT CONDITIONS //
	MesCP_Read 					:= TRUE  ; 
	
// METHODS CALLS //
	IF bInit THEN
		M_Init() ; 
		bInit							:= FALSE ; 
	ELSIF CmdInit_G OR IN_CmdReset_L THEN 
		bInit:= TRUE ;
	END_IF

	M_Read() ; 	
	M_AlarmManagement();
END_METHOD

METHOD M_Init
VAR 

END_VAR
	
AX_Quantity[1] := 12;
AX_Quantity[2] := 18;
AX_Quantity[3] := 32;
AX_Quantity[4] := 4;
AX_Quantity[5] := 32;

AX_Address[1]  := 2999;
AX_Address[2]  := 3020;
AX_Address[3]  := 3053;
AX_Address[4]  := 3107;
AX_Address[5]  := 3203;
END_METHOD

METHOD M_Read
//////////////////
//  Read Modbus Variable for PCS . 
/////////////////
VAR 
	// Method local variables (reinitialized at each cycle) 
	MW 					: FB_MergeWordsToFloat; 
	KK					: BYTE;  						// FOR Loop 
	MW2					: FB_MergeWordsToDint ; 

	
END_VAR
// CP-Read / Write 

MesDataExd.MesData.MesCP_Read := MesCP_Read ; 
 

IF MesCP_Read  THEN	

RTrigI(CLK:= ClockRead AND MesCP_Read);
//Metrology
FOR KK:=1 TO 5 DO  
	InputStructRead[KK].InBuffer := ADR(MesBlock_Temp[KK]);
	InputStructRead[KK].InFunction := 3;
	InputStructRead[KK].InQuantity := AX_Quantity[KK];
	InputStructRead[KK].InStartAddr := AX_Address[KK];
	InputStructRead[KK].InUnitID := ParamUnitID;
	
	InputStructRead[KK].OutBusy := ADR(Busy);
	InputStructRead[KK].OutError := ADR(OutErrorMbRead[KK]);
	//InputStructRead[KK].OutCompleted := ADR(bReadCompleted);
	
	IF RTrigI.Q THEN 
		A1_SUBMV.FB_ModbusReadRTU.M_AddAction_FIFO(InStruct:= InputStructRead[KK] , InPriority:=1 ) ; 
	END_IF
	
END_FOR 
// PROPERTIES UPDATE // 
	// Block 1
//MW( WORD_STRONG:= MesBlock_Temp[1][1], 	WORD_WEAK := MesBlock_Temp[1][2],	SIGNED:=TRUE, FIX:=0 , SIZE:=2, VAR_OUT := MesDataExd.MesData.MesI2);
	

MW( WORD_STRONG:= MesBlock_Temp[1][1], 	WORD_WEAK := MesBlock_Temp[1][2], VAR_OUT := MesDataExd.MesData.MesI1);
MW( WORD_STRONG:= MesBlock_Temp[1][3], 	WORD_WEAK := MesBlock_Temp[1][4], VAR_OUT:= MesDataExd.MesData.MesI2);
MW( WORD_STRONG:= MesBlock_Temp[1][5], 	WORD_WEAK := MesBlock_Temp[1][6], VAR_OUT:= MesDataExd.MesData.MesI3);
MW( WORD_STRONG:= MesBlock_Temp[1][7], 	WORD_WEAK := MesBlock_Temp[1][8], VAR_OUT:= MesDataExd.MesData.MesIN);
MW( WORD_STRONG:= MesBlock_Temp[1][11], 	WORD_WEAK := MesBlock_Temp[1][12], VAR_OUT:= MesDataExd.MesData.MesI);

MW(WORD_WEAK := MesBlock_Temp[2][1], 	WORD_STRONG:= MesBlock_Temp[2][2], VAR_OUT:= MesDataExd.MesData.MesU12);		
MW(WORD_WEAK := MesBlock_Temp[2][3], 	WORD_STRONG:= MesBlock_Temp[2][4], VAR_OUT:= MesDataExd.MesData.MesU23);
MW(WORD_WEAK := MesBlock_Temp[2][5], 	WORD_STRONG:= MesBlock_Temp[2][6], VAR_OUT:= MesDataExd.MesData.MesU31);
MW(WORD_WEAK := MesBlock_Temp[2][7], 	WORD_STRONG:= MesBlock_Temp[2][8], VAR_OUT:= MesDataExd.MesData.MesU);		// Seule donnée valide en monophasée. Il faut d'ailleur inverser les words strongs et word weak quand on passe le settings de triphasé à monophasé . 
MW(WORD_WEAK := MesBlock_Temp[2][9], 	WORD_STRONG:= MesBlock_Temp[2][10], VAR_OUT:= MesDataExd.MesData.MesV1);
MW(WORD_WEAK := MesBlock_Temp[2][11], WORD_STRONG := MesBlock_Temp[2][12], VAR_OUT:= MesDataExd.MesData.MesV2);
MW(WORD_WEAK := MesBlock_Temp[2][13], WORD_STRONG := MesBlock_Temp[2][14], VAR_OUT:= MesDataExd.MesData.MesV3);
MW(WORD_WEAK := MesBlock_Temp[2][17], WORD_STRONG := MesBlock_Temp[2][18], VAR_OUT:= MesDataExd.MesData.MesV);

MW( WORD_STRONG:= MesBlock_Temp[3][1], 	WORD_WEAK := MesBlock_Temp[3][2], VAR_OUT:= MesDataExd.MesData.MesP1);
MW( WORD_STRONG:= MesBlock_Temp[3][3], 	WORD_WEAK := MesBlock_Temp[3][4], VAR_OUT:= MesDataExd.MesData.MesP2);
MW( WORD_STRONG:= MesBlock_Temp[3][5], 	WORD_WEAK := MesBlock_Temp[3][6], VAR_OUT:= MesDataExd.MesData.MesP3);
MW( WORD_STRONG:= MesBlock_Temp[3][7], 	WORD_WEAK := MesBlock_Temp[3][8], VAR_OUT:= MesDataExd.MesData.MesP);

MW( WORD_STRONG:= MesBlock_Temp[3][9], 	WORD_WEAK := MesBlock_Temp[3][10], VAR_OUT:= MesDataExd.MesData.MesQ1);
MW( WORD_STRONG:= MesBlock_Temp[3][11], 	WORD_WEAK := MesBlock_Temp[3][12], VAR_OUT:= MesDataExd.MesData.MesQ2);
MW( WORD_STRONG:= MesBlock_Temp[3][13], 	WORD_WEAK := MesBlock_Temp[3][14], VAR_OUT:= MesDataExd.MesData.MesQ3);
MW( WORD_STRONG:= MesBlock_Temp[3][15], 	WORD_WEAK := MesBlock_Temp[3][16], VAR_OUT:= MesDataExd.MesData.MesQ);
MW( WORD_STRONG:= MesBlock_Temp[3][23], 	WORD_WEAK := MesBlock_Temp[3][24], VAR_OUT:= MesDataExd.MesData.MesS);

MW( WORD_STRONG:= MesBlock_Temp[4][1], 	WORD_WEAK := MesBlock_Temp[4][2], VAR_OUT:= MesDataExd.MesData.MesTanPhi);
MW( WORD_STRONG:= MesBlock_Temp[4][3], 	WORD_WEAK := MesBlock_Temp[4][4], VAR_OUT:= MesDataExd.MesData.MesFreq);

MW2( WORD_STRONG:= MesBlock_Temp[5][3], 	WORD_WEAK := MesBlock_Temp[5][4], VAR_OUT := MesDataExd.MesData.MesEActCons,SIZE:=2,FIX:=3);
MW2( WORD_STRONG:= MesBlock_Temp[5][7], 	WORD_WEAK := MesBlock_Temp[5][8], VAR_OUT := MesDataExd.MesData.MesEActProd,SIZE:=2,FIX:=3);
MW2( WORD_STRONG:= MesBlock_Temp[5][19], 	WORD_WEAK := MesBlock_Temp[5][20], VAR_OUT := MesDataExd.MesData.MesEReactProd,SIZE:=2,FIX:=3);
MW2( WORD_STRONG:= MesBlock_Temp[5][23], 	WORD_WEAK := MesBlock_Temp[5][24], VAR_OUT := MesDataExd.MesData.MesEReactCons,SIZE:=2,FIX:=3);


//MW( WORD_STRONG:= MesBlock_Temp[4][3], 	WORD_WEAK := MesBlock_Temp[4][4],	SIGNED:=TRUE, FIX:=0 , SIZE:=2, VAR_OUT := MesDataExd.MesData.MesFreq);
//MW( WORD_STRONG:= MesBlock_Temp[5][1], 	WORD_WEAK := MesBlock_Temp[5][2],	SIGNED:=TRUE, FIX:=0 , SIZE:=2, VAR_OUT := MesDataExd.MesData.MesEActProd);
//MW( WORD_STRONG:= MesBlock_Temp[5][3], 	WORD_WEAK := MesBlock_Temp[5][4],	SIGNED:=TRUE, FIX:=0 , SIZE:=2, VAR_OUT := MesDataExd.MesData.MesEActCons);
//MW( WORD_STRONG:= MesBlock_Temp[5][5], 	WORD_WEAK := MesBlock_Temp[5][6],	SIGNED:=TRUE, FIX:=0 , SIZE:=2, VAR_OUT := MesDataExd.MesData.MesEReactProd);
//MW( WORD_STRONG:= MesBlock_Temp[5][7], 	WORD_WEAK := MesBlock_Temp[5][8],	SIGNED:=TRUE, FIX:=0 , SIZE:=2, VAR_OUT := MesDataExd.MesData.MesEReactCons);
END_IF
END_METHOD

END_FUNCTION_BLOCK

// ---- 01_Equipement_Library/Datalogger/FB_Datalogger_PPCVerrerie.TcPOU
FUNCTION_BLOCK FB_Datalogger_PPCVerrerie	EXTENDS FB_Datalogger_Base	// Data from PPC ( MV + HV )
VAR_INPUT PERSISTENT
	// Parameters of the Object (instance specific) 
	ParamTempoComAlarm			: TIME 			:= T#10S ; 						// (s) Config : Tempo to detect LOC Alarm
	{attribute 'OPC.UA.DA' := '1'} 
	ParamClockReadTime 			: TIME 			:= TIME#200MS;	  				// (Time) Read Modbus Frequency.  
	ParamTimeout				: TIME  		:= T#2S ;			  			// (Time) Timeout for modbus reading
	ParamIPAdr : STRING := '192.168.1.2'; // IP Address for Modbus Requests 
END_VAR
VAR_INPUT
	IN_CmdToggleRead			: BOOL ;
	IN_CmdReset_L				: BOOL  ; // Reset Order .
	
	
	
END_VAR
VAR
MesDataExd	AT %Q*				: Datalogger_PPCVerrerie;
	
	//M_ALARMMANAGEMENT VARIABLES//
	TON_ComAlarm				: TON ; 												// Tempo before detecting loss of communication. 
	TON_ComWarning				: TON ; 												// Tempo before detecting loss of one frame.   
	
	MesComWarning				: BOOL ; 												// True if bad communication .
	
	// M_EXECUTE VARIABLES //
	
	TP1							: TP ; 												// (NA) Tempo to define Modbus Reading Frequency  
	
    Trig_Cmd_Read				: R_TRIG;                       

	// Modbus Read Variables
	
	FB_ModbusReadAI : ARRAY[1..2] OF FB_ModbusRead;
	FB_ModbusReadDI : ARRAY[1..2] OF FB_ModbusReadCoils;
	
	ClockRead					AT %Q*		: BOOL ;
	
	// Temp Blocks Filled by Requests
	
	AI_List_1 				: ARRAY[1..128] OF WORD;
	AI_List_2 				: ARRAY[1..128] OF WORD;
	DI_List_1 				: ARRAY[1..2048] OF BOOL;
	DI_List_2 				: ARRAY[1..2048] OF BOOL;
	
	
	
END_VAR

METHOD M_AlarmManagement : BOOL
VAR_INPUT
END_VAR
//////////////////
// Digiware measurement tool alarm and warning management
/////////////////

VAR 
	// Method local variables (reinitialized at each cycle) 
	FB_AlarmCodeManager			: FB_AlarmCodeManager ; 
	
	ComWarning					: BOOL;			// Error in one of the Modbus Requests
	ComAlarm					: BOOL;			// Error in all Modbus Requests
	
END_VAR
ComWarning 	:= FB_ModbusReadAI[1].ModbusReadAlarm OR FB_ModbusReadAI[2].ModbusReadAlarm OR FB_ModbusReadDI[1].ModbusReadAlarm OR FB_ModbusReadDI[2].ModbusReadAlarm;
ComAlarm 	:= FB_ModbusReadAI[1].ModbusReadAlarm AND FB_ModbusReadAI[2].ModbusReadAlarm AND FB_ModbusReadDI[1].ModbusReadAlarm AND FB_ModbusReadDI[2].ModbusReadAlarm;
	
TON_ComAlarm(IN:= ComAlarm , PT:= ParamTempoComAlarm, Q= MesDataExd.MesData.MesAlarmCom) ;	
TON_ComWarning(IN:= ComWarning  , PT:= ParamTempoComAlarm, Q=>MesComWarning) ;

//	General com alarm : All the read FB fucked up


// ALARM CODES //
	FB_AlarmCodeManager(
		bAlarm1			:= MesDataExd.MesData.MesAlarmCom , 						// Communication Alarm #COM
		bAlarm2			:= MesDataExd.MesData.Transfo_225kV.MesWarning_TempLevel1,	// Transfo_225kV : Img Therm 1
		bAlarm3			:= MesDataExd.MesData.Transfo_225kV.MesWarning_TempLevel2,	// Transfo_225kV : Img Therm 2
		bAlarm4			:= MesDataExd.MesData.Transfo_225kV.MesDataExd.MesData.MesAlarmTemp,	// Transfo_225kV : Trigger Temp Oil
		bAlarm5			:= MesDataExd.MesData.Transfo_225kV.MesAlarm_TapChanger ,	// Transfo 225kV : Defaillance Regleur
		bAlarm6			:= MesDataExd.MesData.Mes20kVCourNeutCuveTempTrigger,		// 20 kV Courant Neutre Cuve : Temp Trigger
		bAlarm7			:= MesDataExd.MesData.Mes20kVCourNeutCuveGazDischarge,		// 20 kV Courant Neutre Cuve : Gaz Discharge
		bAlarm8			:= MesDataExd.MesData.Mes20kVCourNeutCuvePressure,			// 20 kV Courant Neutre Cuve : Pressure
		bAlarm9			:= MesDataExd.MesData.Transfo_225kV.MesDataExd.MesData.MesAlarmGas,	// Transfo 225kV : Trigger BuchHolz
		bAlarm10		:= MesDataExd.MesData.Transfo_225kV.MesTrigger_Deletion,	// Transfo_225kV : Trigger Deletion
		bAlarm11		:= MesDataExd.MesData.Transfo_225kV.MesAlarm_OilLevel,      // Transfo_225kV : Alarm Oil level
		bAlarm12		:= MesDataExd.MesData.DS.MesAlarmState,          		// DS : Doors Open          
		bAlarm13		:= MesDataExd.MesData.FSS.MesAlarmFire,			        // FSS : Fire Alarm
		bAlarm14		:= MesDataExd.MesData.MesLocalRemoteOperation, 			// Local/Remote Operation
		bAlarm15		:= MesDataExd.MesData.ES.MesAlarmState,         	 	// ES : Emergency Stop			 
		wAlarmCode		=>MesDataExd.MesData.MesAlarmCode1);

	FB_AlarmCodeManager(	
		bAlarm1			:= MesDataExd.MesData.ProtectRelay_Transfo225kV.MesAlarm_DiscordSectLigneHTB,	//	ProtectRelay_Transfo_225kV :	Alarm Discord Sect Ligne HTB
		bAlarm2			:= MesDataExd.MesData.ProtectRelay_Transfo225kV.MesAlarm_DiscordSectMaltHTB ,   //  ProtectRelay_Transfo_225kV : Alarm Discord Sect Malt HTB 
		bAlarm3			:= MesDataExd.MesData.ProtectRelay_Transfo225kV.MesAlarm_DiscordSectDisjHTB ,   //  ProtectRelay_Transfo_225kV : Alarm Discord Sect Disj HTB 
		bAlarm4			:= MesDataExd.MesData.ProtectRelay_Transfo225kV.MesAlarm_TeleCondamne       ,   //  ProtectRelay_Transfo_225kV : Alarm Tele Condamne       
		bAlarm5			:= MesDataExd.MesData.ProtectRelay_Transfo225kV.MesAlarm_DeTeleCondamne     ,   //  ProtectRelay_Transfo_225kV : Alarm DeTele Condamne     
		bAlarm6			:= MesDataExd.MesData.ProtectRelay_Transfo225kV.MesAlarm_DiscordTeleCondamne,   //  ProtectRelay_Transfo_225kV : Alarm Discord Tele Condamne
		bAlarm7			:= MesDataExd.MesData.ProtectRelay_Transfo225kV.MesDataExd.MesData.MesAlarmImax        ,   //  ProtectRelay_Transfo_225kV : Alarm Imax
		bAlarm8			:= MesDataExd.MesData.ProtectRelay_Transfo225kV.MesAlarm_IoMaxCoteProd      ,   //  ProtectRelay_Transfo_225kV : Alarm Io Max Cote Prod
		bAlarm9			:= MesDataExd.MesData.ProtectRelay_Transfo225kV.MesDataExd.MesData.MesAlarmUmin        ,   //  ProtectRelay_Transfo_225kV : Alarm U min
		bAlarm10		:= MesDataExd.MesData.ProtectRelay_Transfo225kV.MesDataExd.MesData.MesAlarmUmin_Long   ,   //  ProtectRelay_Transfo_225kV : Alarm U min Long
		bAlarm11		:= MesDataExd.MesData.ProtectRelay_Transfo225kV.MesAlarmUMax                ,   //  ProtectRelay_Transfo_225kV : Alarm U max
		bAlarm12		:= MesDataExd.MesData.ProtectRelay_Transfo225kV.MesAlarmUMax_Long           ,   //  ProtectRelay_Transfo_225kV : Alarm U max Long
		bAlarm13		:= MesDataExd.MesData.ProtectRelay_Transfo225kV.MesAlarm_PhaseRpt           ,   //  ProtectRelay_Transfo_225kV : Alarm Phase Rpt
		bAlarm14		:= MesDataExd.MesData.ProtectRelay_Transfo225kV.MesAlarm_ImgTherm     		,	//	ProtectRelay_Transfo_225kV : Alarm Img Therm
		bAlarm15		:= MesDataExd.MesData.ProtectRelay_Transfo225kV.MesAlarm_DifferTransfo		,	//  ProtectRelay_Transfo_225kV : Alarm Differ Transfo
		wAlarmCode		=>MesDataExd.MesData.MesAlarmCode2);	


	FB_AlarmCodeManager(	
		bAlarm1			:= MesDataExd.MesData.ProtectRelay_Transfo225kV.MesAlarm_FreqMax ,	// ProtectRelay_Transfo_225kV : Alarm Freq Max
		bAlarm2			:= MesDataExd.MesData.ProtectRelay_Transfo225kV.MesAlarm_FreqMin ,  // ProtectRelay_Transfo_225kV : Alarm Freq Min
		bAlarm3			:= MesDataExd.MesData.MainHVCB.MesDataExd.MesData.MesClosed ,					// MainHVCB : Closed 
		bAlarm4			:= MesDataExd.MesData.MainHVCB.MesAlarm_SF6      ,					// MainHVCB : Alarm SF6
		bAlarm5			:= MesDataExd.MesData.MainHVCB.MesAlarm_Disarmed ,					// MainHVCB : Alarm Disarmed
		bAlarm6			:= MesDataExd.MesData.MainHVCB.MesComutLocal     ,					// MainHVCB : Comut Local
		bAlarm7			:= MesDataExd.MesData.Transfo_225kV.MesTransfoRefrigLocal,    		// Transfo_225kV : Transfo Refrig Local
		bAlarm8			:= MesDataExd.MesData.Transfo_225kV.MesTrigger_NonReturnValve,      // Transfo_225kV : Trigger Non Return Valve
		bAlarm9			:= MesDataExd.MesData.Transfo_225kV.MesTrigger_ProtectRelay,        // Transfo_225kV : Trigger Protect Relay
		bAlarm10		:= MesDataExd.MesData.Transfo_Aux.MesDataExd.MesData.MesAlarmTemp,				// Transfo_Aux : Alarm Temp
		bAlarm11		:= MesDataExd.MesData.Transfo_Aux.MesDataExd.MesData.MesAlarmGas,              // Transfo_Aux : Alarm Gas
		bAlarm12		:= MesDataExd.MesData.Transfo_Aux.MesDataExd.MesData.MesAlarmOilLevel,         // Transfo_Aux : Alarm Pressure
		bAlarm13		:= MesDataExd.MesData.MesAuxTransfoMeltingFusesContact,			// Transfo_Aux : Melting Fuses Contact     
		bAlarm14		:= MesDataExd.MesData.MesAuxTransfoSwitchGear,                     // Transfo_Aux : Transfo Switch Gear
		bAlarm15		:=FALSE,
		wAlarmCode		=>MesDataExd.MesData.MesAlarmCode3);			
		
		
// WARNING CODES //
	FB_AlarmCodeManager(		
		bAlarm1			:=MesComWarning	,				 							// Communication Warning
		bAlarm2			:= MesDataExd.MesData.ProtectRelay_MainHVCB.MesAlarm_Phase1 , 			// ProtectRelay_MainHVCB : Default Phase 1       
		bAlarm3			:= MesDataExd.MesData.ProtectRelay_MainHVCB.MesAlarm_Phase2 , 			// ProtectRelay_MainHVCB : Default Phase 2       
		bAlarm4			:= MesDataExd.MesData.ProtectRelay_MainHVCB.MesAlarm_Phase3 , 			// ProtectRelay_MainHVCB : Default Phase 3       
		bAlarm5			:= MesDataExd.MesData.ProtectRelay_MainHVCB.MesAlarm_PhaseRpt , 		// ProtectRelay_MainHVCB : Default Phase Rpt      
		bAlarm6			:= MesDataExd.MesData.ProtectRelay_MainHVCB.MesAlarm_Ground , 			// ProtectRelay_MainHVCB : Default Phase Ground        
		bAlarm7			:= MesDataExd.MesData.ProtectRelay_MainHVCB.MesAlarm_GroundRpt , 		// ProtectRelay_MainHVCB : Default Phase Ground Rpt     
		bAlarm8			:= MesDataExd.MesData.ProtectRelay_MainHVCB.MesAlarm_MaxUInverse , 		// ProtectRelay_MainHVCB : Default Max U Inverse   
		bAlarm9			:= MesDataExd.MesData.ProtectRelay_MainHVCB.MesAlarm_MaxP , 			// ProtectRelay_MainHVCB : Default Max P
		bAlarm10		:= MesDataExd.MesData.ProtectRelay_MainHVCB.MesAlarm_CB , 				// ProtectRelay_MainHVCB : Default Circuit Breaker
		bAlarm11		:= MesDataExd.MesData.ProtectRelay_MainHVCB.MesAlarm_Watchdog , 		// ProtectRelay_MainHVCB : Default Watchdog     
		bAlarm12		:= MesDataExd.MesData.ProtectRelay_MainHVCB.MesDataExd.MesData.MesAlarmTCS  , 		// ProtectRelay_MainHVCB : Default Major        
		bAlarm13		:= MesDataExd.MesData.ProtectRelay_Transfo225kV.MesAlarm_PhaseRpt ,		// ProtectRelay_Transfo225kV : Default Phase Rpt
		bAlarm14		:= MesDataExd.MesData.ProtectRelay_Transfo225kV.MesAlarm_ImgTherm , 	// ProtectRelay_Transfo225kV : Default img Therm
		bAlarm15		:= MesDataExd.MesData.MainHVCB.MesAlarm_ArmingMotor , 					// MainHVCB : Default Arming Motor
		wAlarmCode		=>MesDataExd.MesData.MesWarningCode1);

	FB_AlarmCodeManager(		
		bAlarm1			:= MesDataExd.MesData.MainHVCB.MesAlarm_230V, 							// MainHVCB : Default Aux 230 Vac				 
		bAlarm2			:= MesDataExd.MesData.MainHVCB.MesAlarmPwr, 							// MainHVCB : Default Alim Bobine
		bAlarm3			:= MesDataExd.MesData.Transfo_225kV.MesWarningGas, 						// Transfo_225kV : Buchholz Gas Warning
		bAlarm4			:= MesDataExd.MesData.Transfo_225kV.MesDataExd.MesData.MesWarningTemp, 			// Transfo_225kV : Temperature Warning
		bAlarm5			:= MesDataExd.MesData.ProtectRelay_Transfo225kV.MesDataExd.MesData.MesAlarmTCS , 	// ProtectRelay_Transfo225kV : Major Default
		bAlarm6			:= MesDataExd.MesData.ProtectRelay_Transfo225kV.MesWarning_ImgTherm , 	// ProtectRelay_Transfo225kV : Warning Img Therm
		bAlarm7			:= MesDataExd.MesData.TapChanger.MesAlarm,								// 225 kV Regleur : Default
		bAlarm8			:= MesDataExd.MesData.TapChanger.MesAlarm_Discordance, 					// 225 kV Regleur : Default Discordance
		bAlarm9			:= MesDataExd.MesData.ProtectRelay_MainMVCB.MesAlarm_Phase1, 			// Protection Relay Main MVCB : Default Phase 1
		bAlarm10		:= MesDataExd.MesData.ProtectRelay_MainMVCB.MesAlarm_Phase2, 			// Protection Relay Main MVCB : Default Phase 2
		bAlarm11		:= MesDataExd.MesData.ProtectRelay_MainMVCB.MesAlarm_CB, 				// Protection Relay Main MVCB : Default Circuit Breaker
		bAlarm12		:=FALSE , 													//
		bAlarm13		:= MesDataExd.MesData.MainMVCB.MesTripped 	, 							// Main MVCB : Tripped
		bAlarm14		:= MesDataExd.MesData.ProtectRelay_MainMVCB.MesDataExd.MesData.MesAlarmTCS , 		// Protection Relay Main MVCB : Alarm TCS
		bAlarm15		:= MesDataExd.MesData.ProtectRelay_MainMVCB.MesDataExd.MesData.MesWatchdog,		// Protection Relay Main MVCB : Watchdog
		wAlarmCode		=>MesDataExd.MesData.MesWarningCode2);		

	FB_AlarmCodeManager(		
		bAlarm1			:= MesDataExd.MesData.ProtectRelay_FeederMVCB[1].MesDataExd.MesData.MesAlarmImax, 							//  ProtectRelay_FeederMVCB Midi Max I Alarm
		bAlarm2			:= MesDataExd.MesData.ProtectRelay_FeederMVCB[1].MesAlarm_MaxP ,								//  ProtectRelay_FeederMVCB Midi Max P Alarm 
		bAlarm3			:= MesDataExd.MesData.ProtectRelay_FeederMVCB[1].MesAlarm_Ground , 								//  ProtectRelay_FeederMVCB Midi Ground Alarm
		bAlarm4			:= MesDataExd.MesData.ProtectRelay_FeederMVCB[1].MesAlarm_CablesOvercharge, 					//	ProtectRelay_FeederMVCB Midi Cables Overcharge
		bAlarm5			:= MesDataExd.MesData.ProtectRelay_FeederMVCB[1].MesAlarm_FaultFrom225kV, 						//  ProtectRelay_FeederMVCB Midi Fault From 225 kV   
		bAlarm6			:= MesDataExd.MesData.ProtectRelay_FeederMVCB[1].MesDataExd.MesData.MesAlarmTCS , 							//  ProtectRelay_FeederMVCB Midi Default Major       
		bAlarm7			:= MesDataExd.MesData.ProtectRelay_FeederMVCB[2].MesDataExd.MesData.MesAlarmImax, 	 						//  ProtectRelay_FeederMVCB Plat Max I Alarm      
		bAlarm8			:= MesDataExd.MesData.ProtectRelay_FeederMVCB[2].MesAlarm_MaxP ,			     				//  ProtectRelay_FeederMVCB Plat Max P Alarm        
		bAlarm9			:= MesDataExd.MesData.ProtectRelay_FeederMVCB[2].MesAlarm_Ground , 		   						//  ProtectRelay_FeederMVCB Plat Ground Alarm          
		bAlarm10		:= MesDataExd.MesData.ProtectRelay_FeederMVCB[2].MesAlarm_CablesOvercharge, 					//  ProtectRelay_FeederMVCB Plat Cables Overcharge 
		bAlarm11		:= MesDataExd.MesData.ProtectRelay_FeederMVCB[2].MesAlarm_FaultFrom225kV, 	 					//  ProtectRelay_FeederMVCB Plat Fault From 225 kV    
		bAlarm12		:= MesDataExd.MesData.ProtectRelay_FeederMVCB[2].MesDataExd.MesData.MesAlarmTCS,				 			//  ProtectRelay_FeederMVCB Plat Default Major                  
		bAlarm13		:=FALSE,   //
		bAlarm14		:=FALSE,   //
		bAlarm15		:=FALSE,   //
		wAlarmCode		=>MesDataExd.MesData.MesWarningCode3);

	FB_AlarmCodeManager(		
		bAlarm1			:= MesDataExd.MesData.Mes20kVCourNeutCuveDefaultMasseCuve1,			//	 20 kV Courant Neutre Cuve Default Masse 1
		bAlarm2			:= MesDataExd.MesData.Mes20kVCourNeutCuveDefaultMasseCuve2,			//	 20 kV Courant Neutre Cuve Default Masse 2
		bAlarm3			:= MesDataExd.MesData.Mes20kVCourNeutCuveDefaultGround,				//	 20 kV Courant Neutre Cuve Default Ground 
		bAlarm4			:= MesDataExd.MesData.Mes20kVCourNeutCuveTempAlarm,					//	 20 kV Courant Neutre Cuve Temp  
		bAlarm5			:= MesDataExd.MesData.MesAuxBt400VDefaultPermut, 					//	 Aux Bt 400 V  : Default Permut 
		bAlarm6			:= MesDataExd.MesData.UPS_CE.MesAlarm_Batt, 			      		//	 UPC CE : Default Batt
		bAlarm7			:= MesDataExd.MesData.UPS_CE.MesDataExd.MesData.MesAlarmState, 				//	 UPC CE : Default Redress
		bAlarm8			:= MesDataExd.MesData.UPS_CE.MesAlarm_IsolBatt,		    			//   UPC CE : Default Isol Batt
		bAlarm9			:= MesDataExd.MesData.UPS_TCM.MesAlarm_Batt,			      		//   UPC TCM : Default Batt
		bAlarm10		:= MesDataExd.MesData.UPS_TCM.MesDataExd.MesData.MesAlarmState,	 			//	 UPC TCM : Default Redress
		bAlarm11		:= MesDataExd.MesData.MesAuxBtDefaultInverter, 						//	 Aux Bt : Default Inverter
		bAlarm12		:= MesDataExd.MesData.MesAuxBtSyntDefaultDistrib48VccJdb, 			//	 Aux Bt Synt : Default Distrib 48 Vcc Jdb
		bAlarm13		:= MesDataExd.MesData.MesAuxBtSyntDefaultDistrib48VccLocker, 		//	 Aux Bt Synt : Default Distrib 48 Vcc Locker
		bAlarm14		:=FALSE, //
		bAlarm15		:=FALSE, //
		wAlarmCode		=>MesDataExd.MesData.MesWarningCode4);		
		
	FB_AlarmCodeManager(		
		bAlarm1			:= MesDataExd.MesData.Mes20kVCourNeutCuveMaxIexp2,	//	 20 kV Courant Neutre Cuve Default Max I Exp 2
		bAlarm2			:= MesDataExd.MesData.Mes20kVCourNeutCuveMaxIexp4,  //	 20 kV Courant Neutre Cuve Default Max I Exp 4
		bAlarm3			:= MesDataExd.MesData.Mes20kVCourNeutCuveMaxI0exp4, //	 20 kV Courant Neutre Cuve Default Max I0 Exp 4
		bAlarm4			:= MesDataExd.MesData.ProtectRelay_FeederMVCB[1].MesDataExd.MesData.MesTripped, // ProtectRelay_FeederMVCB Midi Tripped
		bAlarm5			:= MesDataExd.MesData.ProtectRelay_FeederMVCB[2].MesDataExd.MesData.MesTripped, // ProtectRelay_FeederMVCB Plat Tripped
		bAlarm6			:= MesDataExd.MesData.MesAuxHTSect225kV		,					//	Aux HT : Sect 225 kV
		bAlarm7			:= MesDataExd.MesData.MesAuxHtSmaltHTBOpen	,                   //	Aux HT : Malt HTB Open
		bAlarm8			:= MesDataExd.MesData.MesAuxHtFusionFuseMeasures225kV	,       //	Aux HT : Fusion Fuse Measures 225 kV
		bAlarm9			:= MesDataExd.MesData.MesAuxHtFusionFuseProtect225kV	,       //  Aux HT : Fusion Fuse Protect 225 kV
		bAlarm10		:= MesDataExd.MesData.MesAuxHtFusionFuseCountRte225kV	,       //	Aux HT : Fusion Fuse Count Rte 225 kV
		bAlarm11		:= MesDataExd.MesData.MesAuxHtShortCircuitCurrentProtectCcp2,   //  Aux HT : Short Circuit Current Protect Ccp2
		bAlarm12		:= MesDataExd.MesData.MesAuxHtDisjCount20kVOpen		,           //	Aux HT : Disj Count 20kV Open
		bAlarm13		:= MesDataExd.MesData.MesAuxHtDisjRefVoltage20kVOpen,			//  Aux HT : Disj Ref Voltage 20kV Open
		bAlarm14		:= MesDataExd.MesData.MesAuxHtShortCircuitCurrentProtectCcp3, 	//	Aux HT : Short Circuit Current Protect Ccp3
		bAlarm15		:= MesDataExd.MesData.MesAuxBtTriggerGeneralDisj, 				//  Aux BT : Trigger General Disj
		wAlarmCode		=>MesDataExd.MesData.MesWarningCode5);
		
	FB_AlarmCodeManager(		
		bAlarm1			:= MesDataExd.MesData.Mes20kVCourNeutCuveMaxIexp2,	//	 20 kV Courant Neutre Cuve Default Max I Exp 2
		bAlarm2			:= MesDataExd.MesData.Mes20kVCourNeutCuveMaxIexp4,  //	 20 kV Courant Neutre Cuve Default Max I Exp 4
		bAlarm3			:= MesDataExd.MesData.Mes20kVCourNeutCuveMaxI0exp4, //	 20 kV Courant Neutre Cuve Default Max I0 Exp 4
		bAlarm4			:= MesDataExd.MesData.ProtectRelay_FeederMVCB[1].MesDataExd.MesData.MesTripped, // ProtectRelay_FeederMVCB Midi Tripped
		bAlarm5			:= MesDataExd.MesData.ProtectRelay_FeederMVCB[2].MesDataExd.MesData.MesTripped, // ProtectRelay_FeederMVCB Plat Tripped
		bAlarm6			:= MesDataExd.MesData.MesAuxHTSect225kV		,					//	Aux HT : Sect 225 kV
		bAlarm7			:= MesDataExd.MesData.MesAuxHtSmaltHTBOpen	,                   //	Aux HT : Malt HTB Open
		bAlarm8			:= MesDataExd.MesData.MesAuxHtFusionFuseMeasures225kV	,       //	Aux HT : Fusion Fuse Measures 225 kV
		bAlarm9			:= MesDataExd.MesData.MesAuxHtFusionFuseProtect225kV	,       //  Aux HT : Fusion Fuse Protect 225 kV
		bAlarm10		:= MesDataExd.MesData.MesAuxHtFusionFuseCountRte225kV	,       //	Aux HT : Fusion Fuse Count Rte 225 kV
		bAlarm11		:= MesDataExd.MesData.MesAuxHtShortCircuitCurrentProtectCcp2,   //  Aux HT : Short Circuit Current Protect Ccp2
		bAlarm12		:= MesDataExd.MesData.MesAuxHtDisjCount20kVOpen		,           //	Aux HT : Disj Count 20kV Open
		bAlarm13		:= MesDataExd.MesData.MesAuxHtDisjRefVoltage20kVOpen,			//  Aux HT : Disj Ref Voltage 20kV Open
		bAlarm14		:= MesDataExd.MesData.MesAuxHtShortCircuitCurrentProtectCcp3, 	//	Aux HT : Short Circuit Current Protect Ccp3
		bAlarm15		:= MesDataExd.MesData.MesAuxBtTriggerGeneralDisj, 				//  Aux BT : Trigger General Disj
		wAlarmCode		=>MesDataExd.MesData.MesWarningCode6);
		
		
// EVENT CODE //
	FB_AlarmCodeManager(
		bAlarm1			:= MesDataExd.MesData.MesAuxBt400VManqueAC			 ,  		// Aux BT 400 V : Manque AC     
		bAlarm2			:= MesDataExd.MesData.MesAuxBt400VDecltAntenneScada	 ,  		// Aux BT 400 V : Declt Antenne Scada
		bAlarm3			:= MesDataExd.MesData.MesAuxBt400VDecltAntennePrio	 ,  		// Aux BT 400 V : Declt Antenne Prio
		bAlarm4			:= MesDataExd.MesData.MesAuxBt400VVoltageLossNormalAlim	, 		// Aux BT 400 V : Voltage Loss Normal Alim
		bAlarm5			:= MesDataExd.MesData.MesAuxBt400VVoltageLossSecoursAlim,   	// Aux BT 400 V : Voltage Loss Secours Alim
		bAlarm6			:= MesDataExd.MesData.MesAuxBt400VDefaultPermut	,           	// Aux BT 400 V : Default Permut 
		bAlarm7			:= MesDataExd.MesData.TapChanger.MesModeAuto, 					// 225 kV Regleur :	Mode Auto
		bAlarm8			:= MesDataExd.MesData.TapChanger.MesModeManual,                 // 225 kV Regleur :	Mode Manual                                                                                                                                                                                              
		bAlarm9			:= MesDataExd.MesData.TapChanger.MesState_ManoeuverAuthorized, 	// 225 kV Regleur :	State Manoeuver Authorized
		bAlarm10		:= MesDataExd.MesData.TapChanger.MesAlarm_NoOutletDetected, 	// 225 kV Regleur :	No Outlet Detected	
		bAlarm11		:= MesDataExd.MesData.ProtectRelay_MainHVCB.OUT_CmdOpen , 		// ProtectRelay_MainHVCB : Cmd Open
		bAlarm12		:= MesDataExd.MesData.ProtectRelay_MainHVCB.OUT_CmdClose,       // ProtectRelay_MainHVCB : Cmd Close
		bAlarm13		:= MesDataExd.MesData.ProtectRelay_MainMVCB.OUT_CmdOpen ,       // ProtectRelay_MainMVCB : Cmd Open
		bAlarm14		:= MesDataExd.MesData.ProtectRelay_MainMVCB.OUT_CmdClose,       // ProtectRelay_MainMVCB : Cmd Close
		bAlarm15		:=FALSE, 
		wAlarmCode		=>MesDataExd.MesData.MesEventCode1);
	
